LIN {X 0,Y 404.174,Z 269.949,A -85,B 0,C 180,E1 -11024.526,E2 -11024.526} C_VEL
LIN {X 0,Y 404.186,Z 269.95,A -85,B 0,C 180,E1 -11027.302,E2 -11027.302} C_VEL
LIN {X 0,Y 404.143,Z 269.956,A -85,B 0,C 180,E1 -11029.952,E2 -11029.952} C_VEL
LIN {X 0,Y 404.113,Z 269.963,A -85,B 0,C 180,E1 -11033.121,E2 -11033.121} C_VEL
LIN {X 0,Y 404.144,Z 270.047,A -85,B 0,C 180,E1 -11034.335,E2 -11034.335} C_VEL
LIN {X 0,Y 405.121,Z 276.124,A -85,B 0,C 180,E1 -11035.981,E2 -11035.981} C_VEL
LIN {X 0,Y 405.001,Z 280.687,A -85,B 0,C 180,E1 -11037.137,E2 -11037.137} C_VEL
LIN {X 0,Y 408.445,Z 296.726,A -85,B 0,C 180,E1 -11037.6,E2 -11037.6} C_VEL
LIN {X 0,Y 407.757,Z 357.433,A -85,B 0,C 180,E1 -11038.715,E2 -11038.715} C_VEL
LIN {X 0,Y 407.545,Z 367.165,A -85,B 0,C 180,E1 -11039.032,E2 -11039.032} C_VEL
LIN {X 0,Y 407.188,Z 378.033,A -85,B 0,C 180,E1 -11039.56,E2 -11039.56} C_VEL
LIN {X 0,Y 406.752,Z 387.643,A -85,B 0,C 180,E1 -11040.215,E2 -11040.215} C_VEL
LIN {X 0,Y 406.183,Z 396.777,A -85,B 0,C 180,E1 -11041.022,E2 -11041.022} C_VEL
LIN {X 0,Y 405.632,Z 404.168,A -85,B 0,C 180,E1 -11041.827,E2 -11041.827} C_VEL
LIN {X 0,Y 405.183,Z 410.356,A -85,B 0,C 180,E1 -11042.636,E2 -11042.636} C_VEL
LIN {X 0,Y 404.65,Z 417.143,A -85,B 0,C 180,E1 -11043.712,E2 -11043.712} C_VEL
LIN {X 0,Y 404.296,Z 422.137,A -85,B 0,C 180,E1 -11044.668,E2 -11044.668} C_VEL
LIN {X 0,Y 403.869,Z 427.256,A -85,B 0,C 180,E1 -11045.862,E2 -11045.862} C_VEL
LIN {X 0,Y 403.556,Z 430.963,A -85,B 0,C 180,E1 -11046.932,E2 -11046.932} C_VEL
LIN {X 0,Y 403.244,Z 435.139,A -85,B 0,C 180,E1 -11048.531,E2 -11048.531} C_VEL
LIN {X 0,Y 402.977,Z 438.166,A -85,B 0,C 180,E1 -11050.336,E2 -11050.336} C_VEL
LIN {X 0,Y 402.842,Z 439.29,A -85,B 0,C 180,E1 -11051.698,E2 -11051.698} C_VEL
LIN {X 0,Y 402.817,Z 439.578,A -85,B 0,C 180,E1 -11052.747,E2 -11052.747} C_VEL
LIN {X 0,Y 402.872,Z 439.249,A -85,B 0,C 180,E1 -11053.793,E2 -11053.793} C_VEL
LIN {X 0,Y 402.868,Z 438.387,A -85,B 0,C 180,E1 -11054.831,E2 -11054.831} C_VEL
LIN {X 0,Y 402.939,Z 437.007,A -85,B 0,C 180,E1 -11055.866,E2 -11055.866} C_VEL
LIN {X 0,Y 403.162,Z 433.812,A -85,B 0,C 180,E1 -11057.451,E2 -11057.451} C_VEL
LIN {X 0,Y 403.373,Z 429.458,A -85,B 0,C 180,E1 -11058.951,E2 -11058.951} C_VEL
LIN {X 0,Y 403.667,Z 424.469,A -85,B 0,C 180,E1 -11060.227,E2 -11060.227} C_VEL
LIN {X 0,Y 404.026,Z 418.153,A -85,B 0,C 180,E1 -11061.497,E2 -11061.497} C_VEL
LIN {X 0,Y 404.338,Z 412.472,A -85,B 0,C 180,E1 -11062.437,E2 -11062.437} C_VEL
LIN {X 0,Y 404.715,Z 405.485,A -85,B 0,C 180,E1 -11063.394,E2 -11063.394} C_VEL
LIN {X 0,Y 405.091,Z 398.855,A -85,B 0,C 180,E1 -11064.15,E2 -11064.15} C_VEL
LIN {X 0,Y 405.519,Z 390.81,A -85,B 0,C 180,E1 -11064.904,E2 -11064.904} C_VEL
LIN {X 0,Y 405.865,Z 382.508,A -85,B 0,C 180,E1 -11065.531,E2 -11065.531} C_VEL
LIN {X 0,Y 406.085,Z 374.124,A -85,B 0,C 180,E1 -11066.031,E2 -11066.031} C_VEL
LIN {X 0,Y 406.347,Z 364.962,A -85,B 0,C 180,E1 -11066.437,E2 -11066.437} C_VEL
LIN {X 0,Y 406.545,Z 355.549,A -85,B 0,C 180,E1 -11066.717,E2 -11066.717} C_VEL
LIN {X 0,Y 406.925,Z 321.203,A -85,B 0,C 180,E1 -11067.342,E2 -11067.342} C_VEL
LIN {X 0,Y 406.415,Z 315.379,A -85,B 0,C 180,E1 -11067.462,E2 -11067.462} C_VEL
LIN {X 0,Y 403.768,Z 306.003,A -85,B 0,C 180,E1 -11067.712,E2 -11067.712} C_VEL
LIN {X 0,Y 401.116,Z 298.58,A -85,B 0,C 180,E1 -11067.929,E2 -11067.929} C_VEL
LIN {X 0,Y 399.043,Z 290.982,A -85,B 0,C 180,E1 -11068.133,E2 -11068.133} C_VEL
LIN {X 0,Y 397.37,Z 280.75,A -85,B 0,C 180,E1 -11068.385,E2 -11068.385} C_VEL
LIN {X 0,Y 397.583,Z 272.725,A -85,B 0,C 180,E1 -11070.507,E2 -11070.507} C_VEL
LIN {X 0,Y 397.366,Z 270.803,A -85,B 0,C 180,E1 -11071.077,E2 -11071.077} C_VEL
LIN {X 0,Y 397.345,Z 270.804,A -85,B 0,C 180,E1 -11073.042,E2 -11073.042} C_VEL
LIN {X 0,Y 397.319,Z 270.807,A -85,B 0,C 180,E1 -11077.113,E2 -11077.113} C_VEL
LIN {X 0,Y 397.182,Z 270.819,A -85,B 0,C 180,E1 -11080.192,E2 -11080.192} C_VEL
LIN {X 0,Y 397.192,Z 270.825,A -85,B 0,C 180,E1 -11083.322,E2 -11083.322} C_VEL
LIN {X 0,Y 397.148,Z 270.828,A -85,B 0,C 180,E1 -11087.157,E2 -11087.157} C_VEL
LIN {X 0,Y 397.075,Z 270.833,A -85,B 0,C 180,E1 -11090.732,E2 -11090.732} C_VEL
LIN {X 0,Y 397.091,Z 270.831,A -85,B 0,C 180,E1 -11094.021,E2 -11094.021} C_VEL
LIN {X 0,Y 397.061,Z 270.837,A -85,B 0,C 180,E1 -11097.759,E2 -11097.759} C_VEL
LIN {X 0,Y 397.048,Z 270.836,A -85,B 0,C 180,E1 -11100.885,E2 -11100.885} C_VEL
LIN {X 0,Y 397.097,Z 270.829,A -85,B 0,C 180,E1 -11104.496,E2 -11104.496} C_VEL
LIN {X 0,Y 397.065,Z 270.834,A -85,B 0,C 180,E1 -11108.28,E2 -11108.28} C_VEL
LIN {X 0,Y 397.033,Z 270.841,A -85,B 0,C 180,E1 -11111.981,E2 -11111.981} C_VEL
LIN {X 0,Y 397.064,Z 270.835,A -85,B 0,C 180,E1 -11115.073,E2 -11115.073} C_VEL
LIN {X 0,Y 397.045,Z 270.839,A -85,B 0,C 180,E1 -11118.025,E2 -11118.025} C_VEL
LIN {X 0,Y 397.106,Z 270.829,A -85,B 0,C 180,E1 -11121.143,E2 -11121.143} C_VEL
LIN {X 0,Y 397.102,Z 270.83,A -85,B 0,C 180,E1 -11124.501,E2 -11124.501} C_VEL
LIN {X 0,Y 397.064,Z 270.84,A -85,B 0,C 180,E1 -11127.932,E2 -11127.932} C_VEL
LIN {X 0,Y 397.105,Z 270.831,A -85,B 0,C 180,E1 -11130.299,E2 -11130.299} C_VEL
LIN {X 0,Y 397.083,Z 270.836,A -85,B 0,C 180,E1 -11133.743,E2 -11133.743} C_VEL
LIN {X 0,Y 397.094,Z 270.831,A -85,B 0,C 180,E1 -11137.089,E2 -11137.089} C_VEL
LIN {X 0,Y 397.141,Z 270.827,A -85,B 0,C 180,E1 -11140.357,E2 -11140.357} C_VEL
LIN {X 0,Y 397.248,Z 270.921,A -85,B 0,C 180,E1 -11142.721,E2 -11142.721} C_VEL
LIN {X 0,Y 397.144,Z 279.933,A -85,B 0,C 180,E1 -11145.005,E2 -11145.005} C_VEL
LIN {X 0,Y 399.627,Z 297.894,A -85,B 0,C 180,E1 -11145.49,E2 -11145.49} C_VEL
LIN {X 0,Y 398.723,Z 357.712,A -85,B 0,C 180,E1 -11146.855,E2 -11146.855} C_VEL
LIN {X 0,Y 398.525,Z 367.209,A -85,B 0,C 180,E1 -11147.204,E2 -11147.204} C_VEL
LIN {X 0,Y 398.257,Z 377.066,A -85,B 0,C 180,E1 -11147.713,E2 -11147.713} C_VEL
LIN {X 0,Y 397.95,Z 387.333,A -85,B 0,C 180,E1 -11148.415,E2 -11148.415} C_VEL
LIN {X 0,Y 397.542,Z 397.262,A -85,B 0,C 180,E1 -11149.306,E2 -11149.306} C_VEL
LIN {X 0,Y 397.235,Z 405.182,A -85,B 0,C 180,E1 -11150.199,E2 -11150.199} C_VEL
LIN {X 0,Y 396.884,Z 411.771,A -85,B 0,C 180,E1 -11151.09,E2 -11151.09} C_VEL
LIN {X 0,Y 396.59,Z 418.055,A -85,B 0,C 180,E1 -11152.11,E2 -11152.11} C_VEL
LIN {X 0,Y 396.441,Z 423.135,A -85,B 0,C 180,E1 -11153.1,E2 -11153.1} C_VEL
LIN {X 0,Y 396.217,Z 428.598,A -85,B 0,C 180,E1 -11154.405,E2 -11154.405} C_VEL
LIN {X 0,Y 396.034,Z 433.483,A -85,B 0,C 180,E1 -11155.933,E2 -11155.933} C_VEL
LIN {X 0,Y 395.981,Z 435.892,A -85,B 0,C 180,E1 -11156.951,E2 -11156.951} C_VEL
LIN {X 0,Y 395.905,Z 437.67,A -85,B 0,C 180,E1 -11157.969,E2 -11157.969} C_VEL
LIN {X 0,Y 395.839,Z 438.894,A -85,B 0,C 180,E1 -11158.986,E2 -11158.986} C_VEL
LIN {X 0,Y 395.826,Z 439.592,A -85,B 0,C 180,E1 -11160.003,E2 -11160.003} C_VEL
LIN {X 0,Y 395.863,Z 439.772,A -85,B 0,C 180,E1 -11161.02,E2 -11161.02} C_VEL
LIN {X 0,Y 395.955,Z 439.429,A -85,B 0,C 180,E1 -11162.038,E2 -11162.038} C_VEL
LIN {X 0,Y 396.117,Z 438.507,A -85,B 0,C 180,E1 -11163.054,E2 -11163.054} C_VEL
LIN {X 0,Y 396.429,Z 436.049,A -85,B 0,C 180,E1 -11164.579,E2 -11164.579} C_VEL
LIN {X 0,Y 396.518,Z 433.747,A -85,B 0,C 180,E1 -11165.597,E2 -11165.597} C_VEL
LIN {X 0,Y 396.712,Z 430.771,A -85,B 0,C 180,E1 -11166.615,E2 -11166.615} C_VEL
LIN {X 0,Y 397.14,Z 426.848,A -85,B 0,C 180,E1 -11167.688,E2 -11167.688} C_VEL
LIN {X 0,Y 397.653,Z 420.011,A -85,B 0,C 180,E1 -11169.155,E2 -11169.155} C_VEL
LIN {X 0,Y 398.088,Z 414.112,A -85,B 0,C 180,E1 -11170.171,E2 -11170.171} C_VEL
LIN {X 0,Y 398.67,Z 406.947,A -85,B 0,C 180,E1 -11171.184,E2 -11171.184} C_VEL
LIN {X 0,Y 399.293,Z 398.187,A -85,B 0,C 180,E1 -11172.196,E2 -11172.196} C_VEL
LIN {X 0,Y 399.921,Z 388.436,A -85,B 0,C 180,E1 -11173.08,E2 -11173.08} C_VEL
LIN {X 0,Y 400.428,Z 378.521,A -85,B 0,C 180,E1 -11173.774,E2 -11173.774} C_VEL
LIN {X 0,Y 400.814,Z 369.089,A -85,B 0,C 180,E1 -11174.278,E2 -11174.278} C_VEL
LIN {X 0,Y 401.151,Z 358.396,A -85,B 0,C 180,E1 -11174.687,E2 -11174.687} C_VEL
LIN {X 0,Y 402.704,Z 298.527,A -85,B 0,C 180,E1 -11176.176,E2 -11176.176} C_VEL
LIN {X 0,Y 399.798,Z 286.257,A -85,B 0,C 180,E1 -11176.72,E2 -11176.72} C_VEL
LIN {X 0,Y 398.727,Z 282.083,A -85,B 0,C 180,E1 -11176.943,E2 -11176.943} C_VEL
LIN {X 0,Y 398.602,Z 277.725,A -85,B 0,C 180,E1 -11178.064,E2 -11178.064} C_VEL
LIN {X 0,Y 397.171,Z 270.829,A -85,B 0,C 180,E1 -11179.972,E2 -11179.972} C_VEL
LIN {X 0,Y 397.127,Z 270.833,A -85,B 0,C 180,E1 -11184.021,E2 -11184.021} C_VEL
LIN {X 0,Y 397.102,Z 270.834,A -85,B 0,C 180,E1 -11187.759,E2 -11187.759} C_VEL
LIN {X 0,Y 397.087,Z 270.836,A -85,B 0,C 180,E1 -11190.884,E2 -11190.884} C_VEL
LIN {X 0,Y 397.126,Z 270.832,A -85,B 0,C 180,E1 -11194.496,E2 -11194.496} C_VEL
LIN {X 0,Y 397.101,Z 270.834,A -85,B 0,C 180,E1 -11198.278,E2 -11198.278} C_VEL
LIN {X 0,Y 397.067,Z 270.837,A -85,B 0,C 180,E1 -11201.979,E2 -11201.979} C_VEL
LIN {X 0,Y 397.096,Z 270.832,A -85,B 0,C 180,E1 -11205.07,E2 -11205.07} C_VEL
LIN {X 0,Y 397.07,Z 270.834,A -85,B 0,C 180,E1 -11208.023,E2 -11208.023} C_VEL
LIN {X 0,Y 397.109,Z 270.831,A -85,B 0,C 180,E1 -11211.145,E2 -11211.145} C_VEL
LIN {X 0,Y 397.125,Z 270.83,A -85,B 0,C 180,E1 -11214.498,E2 -11214.498} C_VEL
LIN {X 0,Y 397.086,Z 270.834,A -85,B 0,C 180,E1 -11217.929,E2 -11217.929} C_VEL
LIN {X 0,Y 397.131,Z 270.829,A -85,B 0,C 180,E1 -11221.457,E2 -11221.457} C_VEL
LIN {X 0,Y 397.233,Z 270.885,A -85,B 0,C 180,E1 -11224.416,E2 -11224.416} C_VEL
LIN {X 0,Y 398.807,Z 280.938,A -85,B 0,C 180,E1 -11226.824,E2 -11226.824} C_VEL
LIN {X 0,Y 398.07,Z 294.332,A -85,B 0,C 180,E1 -11229.862,E2 -11229.862} C_VEL
LIN {X 0,Y 397.236,Z 309.12,A -85,B 0,C 180,E1 -11233.183,E2 -11233.183} C_VEL
LIN {X 0,Y 400.225,Z 328.076,A -85,B 0,C 180,E1 -11233.934,E2 -11233.934} C_VEL
LIN {X 0,Y 401.508,Z 342.829,A -85,B 0,C 180,E1 -11234.415,E2 -11234.415} C_VEL
LIN {X 0,Y 400.145,Z 395.197,A -85,B 0,C 180,E1 -11235.739,E2 -11235.739} C_VEL
LIN {X 0,Y 399.501,Z 407.511,A -85,B 0,C 180,E1 -11236.261,E2 -11236.261} C_VEL
LIN {X 0,Y 399.004,Z 415.953,A -85,B 0,C 180,E1 -11236.763,E2 -11236.763} C_VEL
LIN {X 0,Y 398.483,Z 424.385,A -85,B 0,C 180,E1 -11237.393,E2 -11237.393} C_VEL
LIN {X 0,Y 397.952,Z 432.588,A -85,B 0,C 180,E1 -11238.153,E2 -11238.153} C_VEL
LIN {X 0,Y 397.399,Z 440.44,A -85,B 0,C 180,E1 -11239.04,E2 -11239.04} C_VEL
LIN {X 0,Y 396.78,Z 449.471,A -85,B 0,C 180,E1 -11240.313,E2 -11240.313} C_VEL
LIN {X 0,Y 396.386,Z 456.463,A -85,B 0,C 180,E1 -11241.589,E2 -11241.589} C_VEL
LIN {X 0,Y 396.123,Z 462.075,A -85,B 0,C 180,E1 -11242.866,E2 -11242.866} C_VEL
LIN {X 0,Y 395.87,Z 467.423,A -85,B 0,C 180,E1 -11244.396,E2 -11244.396} C_VEL
LIN {X 0,Y 395.822,Z 471.467,A -85,B 0,C 180,E1 -11245.927,E2 -11245.927} C_VEL
LIN {X 0,Y 395.822,Z 473.455,A -85,B 0,C 180,E1 -11246.946,E2 -11246.946} C_VEL
LIN {X 0,Y 395.887,Z 474.938,A -85,B 0,C 180,E1 -11247.965,E2 -11247.965} C_VEL
LIN {X 0,Y 395.835,Z 475.884,A -85,B 0,C 180,E1 -11248.982,E2 -11248.982} C_VEL
LIN {X 0,Y 395.824,Z 476.239,A -85,B 0,C 180,E1 -11250,E2 -11250} C_VEL
LIN {X 0,Y 395.825,Z 476.118,A -85,B 0,C 180,E1 -11251.017,E2 -11251.017} C_VEL
LIN {X 0,Y 395.863,Z 475.535,A -85,B 0,C 180,E1 -11252.035,E2 -11252.035} C_VEL
LIN {X 0,Y 395.785,Z 474.474,A -85,B 0,C 180,E1 -11253.053,E2 -11253.053} C_VEL
LIN {X 0,Y 395.881,Z 471.773,A -85,B 0,C 180,E1 -11254.582,E2 -11254.582} C_VEL
LIN {X 0,Y 395.873,Z 469.352,A -85,B 0,C 180,E1 -11255.603,E2 -11255.603} C_VEL
LIN {X 0,Y 396.138,Z 464.417,A -85,B 0,C 180,E1 -11257.134,E2 -11257.134} C_VEL
LIN {X 0,Y 396.439,Z 459.13,A -85,B 0,C 180,E1 -11258.41,E2 -11258.41} C_VEL
LIN {X 0,Y 396.839,Z 453.959,A -85,B 0,C 180,E1 -11259.428,E2 -11259.428} C_VEL
LIN {X 0,Y 397.316,Z 447.75,A -85,B 0,C 180,E1 -11260.446,E2 -11260.446} C_VEL
LIN {X 0,Y 397.808,Z 441.234,A -85,B 0,C 180,E1 -11261.335,E2 -11261.335} C_VEL
LIN {X 0,Y 398.374,Z 433.361,A -85,B 0,C 180,E1 -11262.222,E2 -11262.222} C_VEL
LIN {X 0,Y 399.005,Z 425.058,A -85,B 0,C 180,E1 -11262.978,E2 -11262.978} C_VEL
LIN {X 0,Y 399.684,Z 414.494,A -85,B 0,C 180,E1 -11263.732,E2 -11263.732} C_VEL
LIN {X 0,Y 400.244,Z 402.924,A -85,B 0,C 180,E1 -11264.303,E2 -11264.303} C_VEL
LIN {X 0,Y 400.662,Z 393.87,A -85,B 0,C 180,E1 -11264.601,E2 -11264.601} C_VEL
LIN {X 0,Y 401.065,Z 364.271,A -85,B 0,C 180,E1 -11265.172,E2 -11265.172} C_VEL
LIN {X 0,Y 401.215,Z 341.462,A -85,B 0,C 180,E1 -11265.592,E2 -11265.592} C_VEL
LIN {X 0,Y 399.203,Z 325.467,A -85,B 0,C 180,E1 -11265.99,E2 -11265.99} C_VEL
LIN {X 0,Y 397.495,Z 314.886,A -85,B 0,C 180,E1 -11266.295,E2 -11266.295} C_VEL
LIN {X 0,Y 398.489,Z 298.029,A -85,B 0,C 180,E1 -11270.115,E2 -11270.115} C_VEL
LIN {X 0,Y 399.419,Z 284.203,A -85,B 0,C 180,E1 -11273.296,E2 -11273.296} C_VEL
LIN {X 0,Y 398.417,Z 277.116,A -85,B 0,C 180,E1 -11275.046,E2 -11275.046} C_VEL
LIN {X 0,Y 397.187,Z 270.824,A -85,B 0,C 180,E1 -11276.679,E2 -11276.679} C_VEL
LIN {X 0,Y 397.109,Z 270.829,A -85,B 0,C 180,E1 -11279.863,E2 -11279.863} C_VEL
LIN {X 0,Y 397.119,Z 270.83,A -85,B 0,C 180,E1 -11283.272,E2 -11283.272} C_VEL
LIN {X 0,Y 397.104,Z 270.829,A -85,B 0,C 180,E1 -11286.994,E2 -11286.994} C_VEL
LIN {X 0,Y 397.085,Z 270.833,A -85,B 0,C 180,E1 -11290.44,E2 -11290.44} C_VEL
LIN {X 0,Y 397.108,Z 270.831,A -85,B 0,C 180,E1 -11293.647,E2 -11293.647} C_VEL
LIN {X 0,Y 397.108,Z 270.829,A -85,B 0,C 180,E1 -11296.52,E2 -11296.52} C_VEL
LIN {X 0,Y 397.094,Z 270.828,A -85,B 0,C 180,E1 -11300.418,E2 -11300.418} C_VEL
LIN {X 0,Y 397.104,Z 270.83,A -85,B 0,C 180,E1 -11303.003,E2 -11303.003} C_VEL
LIN {X 0,Y 397.125,Z 270.827,A -85,B 0,C 180,E1 -11306.28,E2 -11306.28} C_VEL
LIN {X 0,Y 397.107,Z 270.831,A -85,B 0,C 180,E1 -11310.135,E2 -11310.135} C_VEL
LIN {X 0,Y 397.102,Z 270.829,A -85,B 0,C 180,E1 -11313.737,E2 -11313.737} C_VEL
LIN {X 0,Y 397.11,Z 270.829,A -85,B 0,C 180,E1 -11317.083,E2 -11317.083} C_VEL
LIN {X 0,Y 397.152,Z 270.824,A -85,B 0,C 180,E1 -11320.35,E2 -11320.35} C_VEL
LIN {X 0,Y 397.171,Z 270.818,A -85,B 0,C 180,E1 -11323.551,E2 -11323.551} C_VEL
LIN {X 0,Y 397.233,Z 270.811,A -85,B 0,C 180,E1 -11326.7,E2 -11326.7} C_VEL
LIN {X 0,Y 397.22,Z 270.809,A -85,B 0,C 180,E1 -11329.806,E2 -11329.806} C_VEL
LIN {X 0,Y 397.352,Z 270.793,A -85,B 0,C 180,E1 -11332.885,E2 -11332.885} C_VEL
LIN {X 0,Y 397.25,Z 270.802,A -85,B 0,C 180,E1 -11334.922,E2 -11334.922} C_VEL
LIN {X 0,Y 397.446,Z 270.789,A -85,B 0,C 180,E1 -11337.97,E2 -11337.97} C_VEL
LIN {X 0,Y 397.575,Z 270.765,A -85,B 0,C 180,E1 -11339.997,E2 -11339.997} C_VEL
LIN {X 0,Y 397.367,Z 270.794,A -85,B 0,C 180,E1 -11343.038,E2 -11343.038} C_VEL
LIN {X 0,Y 397.314,Z 270.798,A -85,B 0,C 180,E1 -11346.518,E2 -11346.518} C_VEL
LIN {X 0,Y 397.232,Z 270.811,A -85,B 0,C 180,E1 -11349.159,E2 -11349.159} C_VEL
LIN {X 0,Y 397.214,Z 270.818,A -85,B 0,C 180,E1 -11352.254,E2 -11352.254} C_VEL
LIN {X 0,Y 397.172,Z 270.816,A -85,B 0,C 180,E1 -11355.388,E2 -11355.388} C_VEL
LIN {X 0,Y 397.152,Z 270.826,A -85,B 0,C 180,E1 -11358.57,E2 -11358.57} C_VEL
LIN {X 0,Y 397.086,Z 270.831,A -85,B 0,C 180,E1 -11361.815,E2 -11361.815} C_VEL
LIN {X 0,Y 397.144,Z 270.823,A -85,B 0,C 180,E1 -11365.128,E2 -11365.128} C_VEL
LIN {X 0,Y 397.148,Z 270.824,A -85,B 0,C 180,E1 -11367.772,E2 -11367.772} C_VEL
LIN {X 0,Y 397.063,Z 270.835,A -85,B 0,C 180,E1 -11370.879,E2 -11370.879} C_VEL
LIN {X 0,Y 397.108,Z 270.829,A -85,B 0,C 180,E1 -11374.49,E2 -11374.49} C_VEL
LIN {X 0,Y 397.082,Z 270.836,A -85,B 0,C 180,E1 -11378.272,E2 -11378.272} C_VEL
LIN {X 0,Y 397.132,Z 270.828,A -85,B 0,C 180,E1 -11381.989,E2 -11381.989} C_VEL
LIN {X 0,Y 397.127,Z 270.832,A -85,B 0,C 180,E1 -11385.056,E2 -11385.056} C_VEL
LIN {X 0,Y 397.131,Z 270.828,A -85,B 0,C 180,E1 -11388.004,E2 -11388.004} C_VEL
LIN {X 0,Y 397.083,Z 270.837,A -85,B 0,C 180,E1 -11391.723,E2 -11391.723} C_VEL
LIN {X 0,Y 397.145,Z 271.028,A -85,B 0,C 180,E1 -11394.113,E2 -11394.113} C_VEL
LIN {X 0,Y 398.139,Z 276.42,A -85,B 0,C 180,E1 -11395.607,E2 -11395.607} C_VEL
LIN {X 0,Y 398.069,Z 280.908,A -85,B 0,C 180,E1 -11396.78,E2 -11396.78} C_VEL
LIN {X 0,Y 401.763,Z 297.882,A -85,B 0,C 180,E1 -11397.299,E2 -11397.299} C_VEL
LIN {X 0,Y 401.021,Z 356.746,A -85,B 0,C 180,E1 -11398.392,E2 -11398.392} C_VEL
LIN {X 0,Y 400.847,Z 365.689,A -85,B 0,C 180,E1 -11398.671,E2 -11398.671} C_VEL
LIN {X 0,Y 400.555,Z 374.511,A -85,B 0,C 180,E1 -11399.071,E2 -11399.071} C_VEL
LIN {X 0,Y 400.146,Z 383.219,A -85,B 0,C 180,E1 -11399.599,E2 -11399.599} C_VEL
LIN {X 0,Y 399.581,Z 392.811,A -85,B 0,C 180,E1 -11400.352,E2 -11400.352} C_VEL
LIN {X 0,Y 398.882,Z 403.425,A -85,B 0,C 180,E1 -11401.45,E2 -11401.45} C_VEL
LIN {X 0,Y 398.239,Z 410.921,A -85,B 0,C 180,E1 -11402.44,E2 -11402.44} C_VEL
LIN {X 0,Y 397.704,Z 417.477,A -85,B 0,C 180,E1 -11403.5,E2 -11403.5} C_VEL
LIN {X 0,Y 397.298,Z 422.771,A -85,B 0,C 180,E1 -11404.538,E2 -11404.538} C_VEL
LIN {X 0,Y 396.886,Z 427.59,A -85,B 0,C 180,E1 -11405.688,E2 -11405.688} C_VEL
LIN {X 0,Y 396.461,Z 432.093,A -85,B 0,C 180,E1 -11407.046,E2 -11407.046} C_VEL
LIN {X 0,Y 396.245,Z 434.867,A -85,B 0,C 180,E1 -11408.132,E2 -11408.132} C_VEL
LIN {X 0,Y 396.046,Z 436.997,A -85,B 0,C 180,E1 -11409.212,E2 -11409.212} C_VEL
LIN {X 0,Y 395.903,Z 438.541,A -85,B 0,C 180,E1 -11410.289,E2 -11410.289} C_VEL
LIN {X 0,Y 395.786,Z 439.51,A -85,B 0,C 180,E1 -11411.36,E2 -11411.36} C_VEL
LIN {X 0,Y 395.742,Z 439.857,A -85,B 0,C 180,E1 -11412.428,E2 -11412.428} C_VEL
LIN {X 0,Y 395.753,Z 439.659,A -85,B 0,C 180,E1 -11413.51,E2 -11413.51} C_VEL
LIN {X 0,Y 395.784,Z 438.964,A -85,B 0,C 180,E1 -11414.553,E2 -11414.553} C_VEL
LIN {X 0,Y 395.846,Z 437.749,A -85,B 0,C 180,E1 -11415.608,E2 -11415.608} C_VEL
LIN {X 0,Y 395.968,Z 435.998,A -85,B 0,C 180,E1 -11416.66,E2 -11416.66} C_VEL
LIN {X 0,Y 396.168,Z 432.139,A -85,B 0,C 180,E1 -11418.229,E2 -11418.229} C_VEL
LIN {X 0,Y 396.47,Z 426.872,A -85,B 0,C 180,E1 -11419.79,E2 -11419.79} C_VEL
LIN {X 0,Y 396.799,Z 421.208,A -85,B 0,C 180,E1 -11421.085,E2 -11421.085} C_VEL
LIN {X 0,Y 397.254,Z 413.626,A -85,B 0,C 180,E1 -11422.432,E2 -11422.432} C_VEL
LIN {X 0,Y 397.692,Z 405.791,A -85,B 0,C 180,E1 -11423.532,E2 -11423.532} C_VEL
LIN {X 0,Y 398.08,Z 399.158,A -85,B 0,C 180,E1 -11424.301,E2 -11424.301} C_VEL
LIN {X 0,Y 398.533,Z 391.104,A -85,B 0,C 180,E1 -11425.068,E2 -11425.068} C_VEL
LIN {X 0,Y 398.879,Z 382.802,A -85,B 0,C 180,E1 -11425.706,E2 -11425.706} C_VEL
LIN {X 0,Y 399.122,Z 374.4,A -85,B 0,C 180,E1 -11426.214,E2 -11426.214} C_VEL
LIN {X 0,Y 399.395,Z 365.22,A -85,B 0,C 180,E1 -11426.627,E2 -11426.627} C_VEL
LIN {X 0,Y 399.598,Z 355.776,A -85,B 0,C 180,E1 -11426.913,E2 -11426.913} C_VEL
LIN {X 0,Y 400.109,Z 296.595,A -85,B 0,C 180,E1 -11427.997,E2 -11427.997} C_VEL
LIN {X 0,Y 399.043,Z 290.982,A -85,B 0,C 180,E1 -11428.133,E2 -11428.133} C_VEL
LIN {X 0,Y 397.721,Z 287.251,A -85,B 0,C 180,E1 -11428.29,E2 -11428.29} C_VEL
LIN {X 0,Y 394.97,Z 283.108,A -85,B 0,C 180,E1 -11428.648,E2 -11428.648} C_VEL
LIN {X 0,Y 392.229,Z 279.677,A -85,B 0,C 180,E1 -11429.148,E2 -11429.148} C_VEL
LIN {X 0,Y 390.853,Z 277.401,A -85,B 0,C 180,E1 -11429.612,E2 -11429.612} C_VEL
LIN {X 0,Y 390.591,Z 276.013,A -85,B 0,C 180,E1 -11429.956,E2 -11429.956} C_VEL
LIN {X 0,Y 390.337,Z 271.679,A -85,B 0,C 180,E1 -11431.161,E2 -11431.161} C_VEL
LIN {X 0,Y 390.279,Z 271.685,A -85,B 0,C 180,E1 -11433.097,E2 -11433.097} C_VEL
LIN {X 0,Y 390.29,Z 271.678,A -85,B 0,C 180,E1 -11436.203,E2 -11436.203} C_VEL
LIN {X 0,Y 390.169,Z 271.699,A -85,B 0,C 180,E1 -11439.33,E2 -11439.33} C_VEL
LIN {X 0,Y 390.16,Z 271.699,A -85,B 0,C 180,E1 -11443.44,E2 -11443.44} C_VEL
LIN {X 0,Y 390.115,Z 271.706,A -85,B 0,C 180,E1 -11447.309,E2 -11447.309} C_VEL
LIN {X 0,Y 390.055,Z 271.707,A -85,B 0,C 180,E1 -11450.472,E2 -11450.472} C_VEL
LIN {X 0,Y 390.034,Z 271.715,A -85,B 0,C 180,E1 -11453.355,E2 -11453.355} C_VEL
LIN {X 0,Y 390.023,Z 271.711,A -85,B 0,C 180,E1 -11456.775,E2 -11456.775} C_VEL
LIN {X 0,Y 390.007,Z 271.713,A -85,B 0,C 180,E1 -11460.303,E2 -11460.303} C_VEL
LIN {X 0,Y 390.041,Z 271.71,A -85,B 0,C 180,E1 -11464.028,E2 -11464.028} C_VEL
LIN {X 0,Y 390.013,Z 271.719,A -85,B 0,C 180,E1 -11467.553,E2 -11467.553} C_VEL
LIN {X 0,Y 389.994,Z 271.714,A -85,B 0,C 180,E1 -11470.818,E2 -11470.818} C_VEL
LIN {X 0,Y 390.031,Z 271.714,A -85,B 0,C 180,E1 -11473.889,E2 -11473.889} C_VEL
LIN {X 0,Y 390.036,Z 271.709,A -85,B 0,C 180,E1 -11476.793,E2 -11476.793} C_VEL
LIN {X 0,Y 390.037,Z 271.714,A -85,B 0,C 180,E1 -11479.564,E2 -11479.564} C_VEL
LIN {X 0,Y 390.024,Z 271.712,A -85,B 0,C 180,E1 -11482.454,E2 -11482.454} C_VEL
LIN {X 0,Y 390.052,Z 271.711,A -85,B 0,C 180,E1 -11486.049,E2 -11486.049} C_VEL
LIN {X 0,Y 390.031,Z 271.717,A -85,B 0,C 180,E1 -11489.874,E2 -11489.874} C_VEL
LIN {X 0,Y 390.043,Z 271.709,A -85,B 0,C 180,E1 -11493.231,E2 -11493.231} C_VEL
LIN {X 0,Y 390.058,Z 271.707,A -85,B 0,C 180,E1 -11496.768,E2 -11496.768} C_VEL
LIN {X 0,Y 390.097,Z 271.708,A -85,B 0,C 180,E1 -11499.987,E2 -11499.987} C_VEL
LIN {X 0,Y 390.195,Z 271.716,A -85,B 0,C 180,E1 -11502.672,E2 -11502.672} C_VEL
LIN {X 0,Y 390.118,Z 280.193,A -85,B 0,C 180,E1 -11504.833,E2 -11504.833} C_VEL
LIN {X 0,Y 392.636,Z 298.37,A -85,B 0,C 180,E1 -11505.333,E2 -11505.333} C_VEL
LIN {X 0,Y 391.685,Z 358.471,A -85,B 0,C 180,E1 -11506.746,E2 -11506.746} C_VEL
LIN {X 0,Y 391.423,Z 369.194,A -85,B 0,C 180,E1 -11507.166,E2 -11507.166} C_VEL
LIN {X 0,Y 391.103,Z 379.735,A -85,B 0,C 180,E1 -11507.749,E2 -11507.749} C_VEL
LIN {X 0,Y 390.777,Z 390.845,A -85,B 0,C 180,E1 -11508.594,E2 -11508.594} C_VEL
LIN {X 0,Y 390.45,Z 398.893,A -85,B 0,C 180,E1 -11509.372,E2 -11509.372} C_VEL
LIN {X 0,Y 390.113,Z 406.617,A -85,B 0,C 180,E1 -11510.28,E2 -11510.28} C_VEL
LIN {X 0,Y 389.683,Z 414.751,A -85,B 0,C 180,E1 -11511.447,E2 -11511.447} C_VEL
LIN {X 0,Y 389.457,Z 421.9,A -85,B 0,C 180,E1 -11512.747,E2 -11512.747} C_VEL
LIN {X 0,Y 389.186,Z 426.546,A -85,B 0,C 180,E1 -11513.783,E2 -11513.783} C_VEL
LIN {X 0,Y 389.099,Z 430.404,A -85,B 0,C 180,E1 -11514.822,E2 -11514.822} C_VEL
LIN {X 0,Y 388.953,Z 433.537,A -85,B 0,C 180,E1 -11515.859,E2 -11515.859} C_VEL
LIN {X 0,Y 388.887,Z 435.986,A -85,B 0,C 180,E1 -11516.896,E2 -11516.896} C_VEL
LIN {X 0,Y 388.823,Z 437.826,A -85,B 0,C 180,E1 -11517.932,E2 -11517.932} C_VEL
LIN {X 0,Y 388.769,Z 439.122,A -85,B 0,C 180,E1 -11518.968,E2 -11518.968} C_VEL
LIN {X 0,Y 388.753,Z 439.893,A -85,B 0,C 180,E1 -11520.003,E2 -11520.003} C_VEL
LIN {X 0,Y 388.792,Z 440.148,A -85,B 0,C 180,E1 -11521.039,E2 -11521.039} C_VEL
LIN {X 0,Y 388.891,Z 439.859,A -85,B 0,C 180,E1 -11522.075,E2 -11522.075} C_VEL
LIN {X 0,Y 389.064,Z 438.964,A -85,B 0,C 180,E1 -11523.11,E2 -11523.11} C_VEL
LIN {X 0,Y 389.393,Z 436.637,A -85,B 0,C 180,E1 -11524.662,E2 -11524.662} C_VEL
LIN {X 0,Y 389.473,Z 432.937,A -85,B 0,C 180,E1 -11526.219,E2 -11526.219} C_VEL
LIN {X 0,Y 390.122,Z 427.786,A -85,B 0,C 180,E1 -11527.768,E2 -11527.768} C_VEL
LIN {X 0,Y 390.583,Z 422.224,A -85,B 0,C 180,E1 -11529.062,E2 -11529.062} C_VEL
LIN {X 0,Y 391.194,Z 415.121,A -85,B 0,C 180,E1 -11530.353,E2 -11530.353} C_VEL
LIN {X 0,Y 391.821,Z 408.122,A -85,B 0,C 180,E1 -11531.382,E2 -11531.382} C_VEL
LIN {X 0,Y 392.377,Z 400.721,A -85,B 0,C 180,E1 -11532.283,E2 -11532.283} C_VEL
LIN {X 0,Y 393.033,Z 391.654,A -85,B 0,C 180,E1 -11533.182,E2 -11533.182} C_VEL
LIN {X 0,Y 393.693,Z 380.651,A -85,B 0,C 180,E1 -11534.014,E2 -11534.014} C_VEL
LIN {X 0,Y 394.101,Z 371.717,A -85,B 0,C 180,E1 -11534.526,E2 -11534.526} C_VEL
LIN {X 0,Y 394.427,Z 361.902,A -85,B 0,C 180,E1 -11534.943,E2 -11534.943} C_VEL
LIN {X 0,Y 395.208,Z 337.111,A -85,B 0,C 180,E1 -11535.598,E2 -11535.598} C_VEL
LIN {X 0,Y 396.254,Z 299.725,A -85,B 0,C 180,E1 -11536.581,E2 -11536.581} C_VEL
LIN {X 0,Y 393.127,Z 286.68,A -85,B 0,C 180,E1 -11537.186,E2 -11537.186} C_VEL
LIN {X 0,Y 391.981,Z 282.688,A -85,B 0,C 180,E1 -11537.389,E2 -11537.389} C_VEL
LIN {X 0,Y 391.731,Z 279.113,A -85,B 0,C 180,E1 -11538.344,E2 -11538.344} C_VEL
LIN {X 0,Y 390.094,Z 271.71,A -85,B 0,C 180,E1 -11540.411,E2 -11540.411} C_VEL
LIN {X 0,Y 390.073,Z 271.708,A -85,B 0,C 180,E1 -11543.355,E2 -11543.355} C_VEL
LIN {X 0,Y 390.062,Z 271.712,A -85,B 0,C 180,E1 -11546.775,E2 -11546.775} C_VEL
LIN {X 0,Y 390.046,Z 271.714,A -85,B 0,C 180,E1 -11550.302,E2 -11550.302} C_VEL
LIN {X 0,Y 390.078,Z 271.709,A -85,B 0,C 180,E1 -11554.026,E2 -11554.026} C_VEL
LIN {X 0,Y 390.047,Z 271.711,A -85,B 0,C 180,E1 -11557.782,E2 -11557.782} C_VEL
LIN {X 0,Y 390.028,Z 271.715,A -85,B 0,C 180,E1 -11560.816,E2 -11560.816} C_VEL
LIN {X 0,Y 390.063,Z 271.707,A -85,B 0,C 180,E1 -11563.887,E2 -11563.887} C_VEL
LIN {X 0,Y 390.065,Z 271.709,A -85,B 0,C 180,E1 -11566.79,E2 -11566.79} C_VEL
LIN {X 0,Y 390.042,Z 271.71,A -85,B 0,C 180,E1 -11569.558,E2 -11569.558} C_VEL
LIN {X 0,Y 390.049,Z 271.714,A -85,B 0,C 180,E1 -11572.451,E2 -11572.451} C_VEL
LIN {X 0,Y 390.078,Z 271.704,A -85,B 0,C 180,E1 -11575.976,E2 -11575.976} C_VEL
LIN {X 0,Y 390.056,Z 271.71,A -85,B 0,C 180,E1 -11579.87,E2 -11579.87} C_VEL
LIN {X 0,Y 390.134,Z 271.7,A -85,B 0,C 180,E1 -11583.233,E2 -11583.233} C_VEL
LIN {X 0,Y 390.174,Z 271.811,A -85,B 0,C 180,E1 -11584.292,E2 -11584.292} C_VEL
LIN {X 0,Y 391.659,Z 280.391,A -85,B 0,C 180,E1 -11586.39,E2 -11586.39} C_VEL
LIN {X 0,Y 391.654,Z 285.495,A -85,B 0,C 180,E1 -11587.584,E2 -11587.584} C_VEL
LIN {X 0,Y 390.625,Z 301.995,A -85,B 0,C 180,E1 -11591.376,E2 -11591.376} C_VEL
LIN {X 0,Y 390.292,Z 307.828,A -85,B 0,C 180,E1 -11592.668,E2 -11592.668} C_VEL
LIN {X 0,Y 393.501,Z 327.282,A -85,B 0,C 180,E1 -11593.469,E2 -11593.469} C_VEL
LIN {X 0,Y 394.986,Z 342.93,A -85,B 0,C 180,E1 -11594.017,E2 -11594.017} C_VEL
LIN {X 0,Y 393.5,Z 394.719,A -85,B 0,C 180,E1 -11595.372,E2 -11595.372} C_VEL
LIN {X 0,Y 392.852,Z 406.868,A -85,B 0,C 180,E1 -11595.892,E2 -11595.892} C_VEL
LIN {X 0,Y 392.147,Z 417.178,A -85,B 0,C 180,E1 -11596.527,E2 -11596.527} C_VEL
LIN {X 0,Y 391.494,Z 426.754,A -85,B 0,C 180,E1 -11597.296,E2 -11597.296} C_VEL
LIN {X 0,Y 390.766,Z 436.713,A -85,B 0,C 180,E1 -11598.326,E2 -11598.326} C_VEL
LIN {X 0,Y 390.173,Z 444.594,A -85,B 0,C 180,E1 -11599.36,E2 -11599.36} C_VEL
LIN {X 0,Y 389.71,Z 451.132,A -85,B 0,C 180,E1 -11600.397,E2 -11600.397} C_VEL
LIN {X 0,Y 389.371,Z 456.569,A -85,B 0,C 180,E1 -11601.436,E2 -11601.436} C_VEL
LIN {X 0,Y 389.127,Z 461.092,A -85,B 0,C 180,E1 -11602.476,E2 -11602.476} C_VEL
LIN {X 0,Y 388.842,Z 465.673,A -85,B 0,C 180,E1 -11603.774,E2 -11603.774} C_VEL
LIN {X 0,Y 388.751,Z 471.069,A -85,B 0,C 180,E1 -11605.853,E2 -11605.853} C_VEL
LIN {X 0,Y 388.724,Z 473.05,A -85,B 0,C 180,E1 -11606.891,E2 -11606.891} C_VEL
LIN {X 0,Y 388.8,Z 474.565,A -85,B 0,C 180,E1 -11607.928,E2 -11607.928} C_VEL
LIN {X 0,Y 388.765,Z 475.519,A -85,B 0,C 180,E1 -11608.964,E2 -11608.964} C_VEL
LIN {X 0,Y 388.751,Z 475.896,A -85,B 0,C 180,E1 -11610,E2 -11610} C_VEL
LIN {X 0,Y 388.756,Z 475.805,A -85,B 0,C 180,E1 -11611.036,E2 -11611.036} C_VEL
LIN {X 0,Y 388.761,Z 475.252,A -85,B 0,C 180,E1 -11612.072,E2 -11612.072} C_VEL
LIN {X 0,Y 388.69,Z 474.213,A -85,B 0,C 180,E1 -11613.109,E2 -11613.109} C_VEL
LIN {X 0,Y 388.791,Z 471.552,A -85,B 0,C 180,E1 -11614.666,E2 -11614.666} C_VEL
LIN {X 0,Y 388.841,Z 467.632,A -85,B 0,C 180,E1 -11616.226,E2 -11616.226} C_VEL
LIN {X 0,Y 389.091,Z 464.267,A -85,B 0,C 180,E1 -11617.264,E2 -11617.264} C_VEL
LIN {X 0,Y 389.393,Z 459.02,A -85,B 0,C 180,E1 -11618.563,E2 -11618.563} C_VEL
LIN {X 0,Y 389.834,Z 453.898,A -85,B 0,C 180,E1 -11619.599,E2 -11619.599} C_VEL
LIN {X 0,Y 390.327,Z 447.75,A -85,B 0,C 180,E1 -11620.635,E2 -11620.635} C_VEL
LIN {X 0,Y 390.861,Z 441.308,A -85,B 0,C 180,E1 -11621.539,E2 -11621.539} C_VEL
LIN {X 0,Y 391.449,Z 433.528,A -85,B 0,C 180,E1 -11622.441,E2 -11622.441} C_VEL
LIN {X 0,Y 392.106,Z 425.344,A -85,B 0,C 180,E1 -11623.21,E2 -11623.21} C_VEL
LIN {X 0,Y 392.706,Z 416.836,A -85,B 0,C 180,E1 -11623.849,E2 -11623.849} C_VEL
LIN {X 0,Y 393.279,Z 406.892,A -85,B 0,C 180,E1 -11624.422,E2 -11624.422} C_VEL
LIN {X 0,Y 393.87,Z 394.279,A -85,B 0,C 180,E1 -11624.896,E2 -11624.896} C_VEL
LIN {X 0,Y 394.26,Z 371.936,A -85,B 0,C 180,E1 -11625.346,E2 -11625.346} C_VEL
LIN {X 0,Y 394.439,Z 341.551,A -85,B 0,C 180,E1 -11625.917,E2 -11625.917} C_VEL
LIN {X 0,Y 392.14,Z 324.021,A -85,B 0,C 180,E1 -11626.369,E2 -11626.369} C_VEL
LIN {X 0,Y 390.555,Z 314.545,A -85,B 0,C 180,E1 -11626.654,E2 -11626.654} C_VEL
LIN {X 0,Y 391.595,Z 297.949,A -85,B 0,C 180,E1 -11630.485,E2 -11630.485} C_VEL
LIN {X 0,Y 392.466,Z 286.357,A -85,B 0,C 180,E1 -11633.201,E2 -11633.201} C_VEL
LIN {X 0,Y 391.838,Z 280.547,A -85,B 0,C 180,E1 -11634.646,E2 -11634.646} C_VEL
LIN {X 0,Y 390.162,Z 271.702,A -85,B 0,C 180,E1 -11636.981,E2 -11636.981} C_VEL
LIN {X 0,Y 390.046,Z 271.71,A -85,B 0,C 180,E1 -11640.299,E2 -11640.299} C_VEL
LIN {X 0,Y 390.077,Z 271.709,A -85,B 0,C 180,E1 -11644.024,E2 -11644.024} C_VEL
LIN {X 0,Y 390.047,Z 271.713,A -85,B 0,C 180,E1 -11647.779,E2 -11647.779} C_VEL
LIN {X 0,Y 390.055,Z 271.71,A -85,B 0,C 180,E1 -11650.818,E2 -11650.818} C_VEL
LIN {X 0,Y 390.061,Z 271.706,A -85,B 0,C 180,E1 -11653.885,E2 -11653.885} C_VEL
LIN {X 0,Y 390.063,Z 271.707,A -85,B 0,C 180,E1 -11656.788,E2 -11656.788} C_VEL
LIN {X 0,Y 390.021,Z 271.716,A -85,B 0,C 180,E1 -11659.554,E2 -11659.554} C_VEL
LIN {X 0,Y 390.047,Z 271.708,A -85,B 0,C 180,E1 -11662.448,E2 -11662.448} C_VEL
LIN {X 0,Y 390.076,Z 271.708,A -85,B 0,C 180,E1 -11665.974,E2 -11665.974} C_VEL
LIN {X 0,Y 390.051,Z 271.709,A -85,B 0,C 180,E1 -11669.868,E2 -11669.868} C_VEL
LIN {X 0,Y 390.061,Z 271.706,A -85,B 0,C 180,E1 -11673.225,E2 -11673.225} C_VEL
LIN {X 0,Y 390.073,Z 271.705,A -85,B 0,C 180,E1 -11676.762,E2 -11676.762} C_VEL
LIN {X 0,Y 390.109,Z 271.703,A -85,B 0,C 180,E1 -11679.981,E2 -11679.981} C_VEL
LIN {X 0,Y 390.143,Z 271.693,A -85,B 0,C 180,E1 -11683.246,E2 -11683.246} C_VEL
LIN {X 0,Y 390.199,Z 271.688,A -85,B 0,C 180,E1 -11686.559,E2 -11686.559} C_VEL
LIN {X 0,Y 390.208,Z 271.685,A -85,B 0,C 180,E1 -11690.668,E2 -11690.668} C_VEL
LIN {X 0,Y 390.327,Z 271.67,A -85,B 0,C 180,E1 -11693.795,E2 -11693.795} C_VEL
LIN {X 0,Y 390.414,Z 271.665,A -85,B 0,C 180,E1 -11697.934,E2 -11697.934} C_VEL
LIN {X 0,Y 390.544,Z 271.641,A -85,B 0,C 180,E1 -11699.997,E2 -11699.997} C_VEL
LIN {X 0,Y 390.302,Z 271.674,A -85,B 0,C 180,E1 -11703.093,E2 -11703.093} C_VEL
LIN {X 0,Y 390.272,Z 271.676,A -85,B 0,C 180,E1 -11706.51,E2 -11706.51} C_VEL
LIN {X 0,Y 390.189,Z 271.688,A -85,B 0,C 180,E1 -11709.325,E2 -11709.325} C_VEL
LIN {X 0,Y 390.165,Z 271.698,A -85,B 0,C 180,E1 -11712.479,E2 -11712.479} C_VEL
LIN {X 0,Y 390.132,Z 271.694,A -85,B 0,C 180,E1 -11715.673,E2 -11715.673} C_VEL
LIN {X 0,Y 390.096,Z 271.702,A -85,B 0,C 180,E1 -11718.918,E2 -11718.918} C_VEL
LIN {X 0,Y 390.03,Z 271.714,A -85,B 0,C 180,E1 -11722.23,E2 -11722.23} C_VEL
LIN {X 0,Y 390.107,Z 271.7,A -85,B 0,C 180,E1 -11725.74,E2 -11725.74} C_VEL
LIN {X 0,Y 390.044,Z 271.71,A -85,B 0,C 180,E1 -11729.106,E2 -11729.106} C_VEL
LIN {X 0,Y 390.026,Z 271.717,A -85,B 0,C 180,E1 -11732.718,E2 -11732.718} C_VEL
LIN {X 0,Y 390.037,Z 271.701,A -85,B 0,C 180,E1 -11735.822,E2 -11735.822} C_VEL
LIN {X 0,Y 390.048,Z 271.708,A -85,B 0,C 180,E1 -11739.215,E2 -11739.215} C_VEL
LIN {X 0,Y 390.097,Z 271.708,A -85,B 0,C 180,E1 -11742.383,E2 -11742.383} C_VEL
LIN {X 0,Y 390.095,Z 271.706,A -85,B 0,C 180,E1 -11745.362,E2 -11745.362} C_VEL
LIN {X 0,Y 390.08,Z 271.708,A -85,B 0,C 180,E1 -11748.193,E2 -11748.193} C_VEL
LIN {X 0,Y 390.069,Z 271.71,A -85,B 0,C 180,E1 -11750.905,E2 -11750.905} C_VEL
LIN {X 0,Y 390.055,Z 271.867,A -85,B 0,C 180,E1 -11753.83,E2 -11753.83} C_VEL
LIN {X 0,Y 391.23,Z 278.559,A -85,B 0,C 180,E1 -11755.715,E2 -11755.715} C_VEL
LIN {X 0,Y 391.19,Z 281.239,A -85,B 0,C 180,E1 -11756.425,E2 -11756.425} C_VEL
LIN {X 0,Y 394.994,Z 298.561,A -85,B 0,C 180,E1 -11756.97,E2 -11756.97} C_VEL
LIN {X 0,Y 394.281,Z 357.432,A -85,B 0,C 180,E1 -11758.088,E2 -11758.088} C_VEL
LIN {X 0,Y 394.049,Z 367.114,A -85,B 0,C 180,E1 -11758.405,E2 -11758.405} C_VEL
LIN {X 0,Y 393.676,Z 377.332,A -85,B 0,C 180,E1 -11758.903,E2 -11758.903} C_VEL
LIN {X 0,Y 393.101,Z 388.628,A -85,B 0,C 180,E1 -11759.683,E2 -11759.683} C_VEL
LIN {X 0,Y 392.46,Z 397.524,A -85,B 0,C 180,E1 -11760.498,E2 -11760.498} C_VEL
LIN {X 0,Y 391.866,Z 405.044,A -85,B 0,C 180,E1 -11761.35,E2 -11761.35} C_VEL
LIN {X 0,Y 391.352,Z 411.066,A -85,B 0,C 180,E1 -11762.166,E2 -11762.166} C_VEL
LIN {X 0,Y 390.764,Z 417.841,A -85,B 0,C 180,E1 -11763.28,E2 -11763.28} C_VEL
LIN {X 0,Y 390.313,Z 423.392,A -85,B 0,C 180,E1 -11764.396,E2 -11764.396} C_VEL
LIN {X 0,Y 389.902,Z 427.937,A -85,B 0,C 180,E1 -11765.508,E2 -11765.508} C_VEL
LIN {X 0,Y 389.531,Z 431.635,A -85,B 0,C 180,E1 -11766.614,E2 -11766.614} C_VEL
LIN {X 0,Y 389.16,Z 435.806,A -85,B 0,C 180,E1 -11768.271,E2 -11768.271} C_VEL
LIN {X 0,Y 388.843,Z 438.696,A -85,B 0,C 180,E1 -11770.012,E2 -11770.012} C_VEL
LIN {X 0,Y 388.726,Z 439.615,A -85,B 0,C 180,E1 -11771.008,E2 -11771.008} C_VEL
LIN {X 0,Y 388.662,Z 440.107,A -85,B 0,C 180,E1 -11772.097,E2 -11772.097} C_VEL
LIN {X 0,Y 388.675,Z 440.014,A -85,B 0,C 180,E1 -11773.385,E2 -11773.385} C_VEL
LIN {X 0,Y 388.687,Z 439.543,A -85,B 0,C 180,E1 -11774.263,E2 -11774.263} C_VEL
LIN {X 0,Y 388.729,Z 438.485,A -85,B 0,C 180,E1 -11775.338,E2 -11775.338} C_VEL
LIN {X 0,Y 388.862,Z 436.811,A -85,B 0,C 180,E1 -11776.411,E2 -11776.411} C_VEL
LIN {X 0,Y 389.058,Z 433.236,A -85,B 0,C 180,E1 -11778.01,E2 -11778.01} C_VEL
LIN {X 0,Y 389.237,Z 430.093,A -85,B 0,C 180,E1 -11779.072,E2 -11779.072} C_VEL
LIN {X 0,Y 389.533,Z 425.102,A -85,B 0,C 180,E1 -11780.393,E2 -11780.393} C_VEL
LIN {X 0,Y 389.95,Z 418.773,A -85,B 0,C 180,E1 -11781.71,E2 -11781.71} C_VEL
LIN {X 0,Y 390.327,Z 412.584,A -85,B 0,C 180,E1 -11782.759,E2 -11782.759} C_VEL
LIN {X 0,Y 390.677,Z 406.095,A -85,B 0,C 180,E1 -11783.674,E2 -11783.674} C_VEL
LIN {X 0,Y 391.097,Z 399.447,A -85,B 0,C 180,E1 -11784.457,E2 -11784.457} C_VEL
LIN {X 0,Y 391.555,Z 391.386,A -85,B 0,C 180,E1 -11785.238,E2 -11785.238} C_VEL
LIN {X 0,Y 391.898,Z 383.079,A -85,B 0,C 180,E1 -11785.887,E2 -11785.887} C_VEL
LIN {X 0,Y 392.167,Z 374.648,A -85,B 0,C 180,E1 -11786.404,E2 -11786.404} C_VEL
LIN {X 0,Y 392.45,Z 365.437,A -85,B 0,C 180,E1 -11786.824,E2 -11786.824} C_VEL
LIN {X 0,Y 392.644,Z 355.957,A -85,B 0,C 180,E1 -11787.115,E2 -11787.115} C_VEL
LIN {X 0,Y 393.133,Z 297.251,A -85,B 0,C 180,E1 -11788.207,E2 -11788.207} C_VEL
LIN {X 0,Y 390.35,Z 281.038,A -85,B 0,C 180,E1 -11788.614,E2 -11788.614} C_VEL
LIN {X 0,Y 390.591,Z 276.013,A -85,B 0,C 180,E1 -11789.956,E2 -11789.956} C_VEL
LIN {X 0,Y 390.337,Z 274.426,A -85,B 0,C 180,E1 -11790.476,E2 -11790.476} C_VEL
LIN {X 0,Y 389.494,Z 273.358,A -85,B 0,C 180,E1 -11791.014,E2 -11791.014} C_VEL
LIN {X 0,Y 386.899,Z 272.409,A -85,B 0,C 180,E1 -11792.113,E2 -11792.113} C_VEL
LIN {X 0,Y 384.234,Z 272.438,A -85,B 0,C 180,E1 -11793.262,E2 -11793.262} C_VEL
LIN {X 0,Y 383.124,Z 272.571,A -85,B 0,C 180,E1 -11794.156,E2 -11794.156} C_VEL
LIN {X 0,Y 383.056,Z 272.579,A -85,B 0,C 180,E1 -11794.459,E2 -11794.459} C_VEL
LIN {X 0,Y 383.247,Z 272.555,A -85,B 0,C 180,E1 -11796.317,E2 -11796.317} C_VEL
LIN {X 0,Y 383.187,Z 272.563,A -85,B 0,C 180,E1 -11798.438,E2 -11798.438} C_VEL
LIN {X 0,Y 383.062,Z 272.581,A -85,B 0,C 180,E1 -11801.643,E2 -11801.643} C_VEL
LIN {X 0,Y 383.075,Z 272.579,A -85,B 0,C 180,E1 -11804.883,E2 -11804.883} C_VEL
LIN {X 0,Y 383.029,Z 272.582,A -85,B 0,C 180,E1 -11808.175,E2 -11808.175} C_VEL
LIN {X 0,Y 382.966,Z 272.595,A -85,B 0,C 180,E1 -11811.533,E2 -11811.533} C_VEL
LIN {X 0,Y 382.986,Z 272.589,A -85,B 0,C 180,E1 -11814.965,E2 -11814.965} C_VEL
LIN {X 0,Y 382.955,Z 272.591,A -85,B 0,C 180,E1 -11818.5,E2 -11818.5} C_VEL
LIN {X 0,Y 382.98,Z 272.589,A -85,B 0,C 180,E1 -11822.153,E2 -11822.153} C_VEL
LIN {X 0,Y 382.99,Z 272.587,A -85,B 0,C 180,E1 -11824.671,E2 -11824.671} C_VEL
LIN {X 0,Y 382.967,Z 272.593,A -85,B 0,C 180,E1 -11827.906,E2 -11827.906} C_VEL
LIN {X 0,Y 382.938,Z 272.597,A -85,B 0,C 180,E1 -11831.354,E2 -11831.354} C_VEL
LIN {X 0,Y 382.972,Z 272.59,A -85,B 0,C 180,E1 -11834.307,E2 -11834.307} C_VEL
LIN {X 0,Y 382.99,Z 272.589,A -85,B 0,C 180,E1 -11837.244,E2 -11837.244} C_VEL
LIN {X 0,Y 382.994,Z 272.588,A -85,B 0,C 180,E1 -11840.418,E2 -11840.418} C_VEL
LIN {X 0,Y 383.008,Z 272.589,A -85,B 0,C 180,E1 -11844.048,E2 -11844.048} C_VEL
LIN {X 0,Y 382.972,Z 272.593,A -85,B 0,C 180,E1 -11847.582,E2 -11847.582} C_VEL
LIN {X 0,Y 382.967,Z 272.593,A -85,B 0,C 180,E1 -11850.303,E2 -11850.303} C_VEL
LIN {X 0,Y 382.993,Z 272.592,A -85,B 0,C 180,E1 -11854.048,E2 -11854.048} C_VEL
LIN {X 0,Y 382.982,Z 272.589,A -85,B 0,C 180,E1 -11857.338,E2 -11857.338} C_VEL
LIN {X 0,Y 383.056,Z 272.58,A -85,B 0,C 180,E1 -11860.72,E2 -11860.72} C_VEL
LIN {X 0,Y 383.173,Z 272.687,A -85,B 0,C 180,E1 -11862.668,E2 -11862.668} C_VEL
LIN {X 0,Y 383.078,Z 280.388,A -85,B 0,C 180,E1 -11864.645,E2 -11864.645} C_VEL
LIN {X 0,Y 385.631,Z 298.483,A -85,B 0,C 180,E1 -11865.162,E2 -11865.162} C_VEL
LIN {X 0,Y 384.635,Z 359.162,A -85,B 0,C 180,E1 -11866.633,E2 -11866.633} C_VEL
LIN {X 0,Y 384.438,Z 368.344,A -85,B 0,C 180,E1 -11866.996,E2 -11866.996} C_VEL
LIN {X 0,Y 384.137,Z 378.025,A -85,B 0,C 180,E1 -11867.523,E2 -11867.523} C_VEL
LIN {X 0,Y 383.827,Z 388.204,A -85,B 0,C 180,E1 -11868.25,E2 -11868.25} C_VEL
LIN {X 0,Y 383.402,Z 398.047,A -85,B 0,C 180,E1 -11869.174,E2 -11869.174} C_VEL
LIN {X 0,Y 383.082,Z 405.949,A -85,B 0,C 180,E1 -11870.1,E2 -11870.1} C_VEL
LIN {X 0,Y 382.631,Z 414.226,A -85,B 0,C 180,E1 -11871.288,E2 -11871.288} C_VEL
LIN {X 0,Y 382.375,Z 421.622,A -85,B 0,C 180,E1 -11872.612,E2 -11872.612} C_VEL
LIN {X 0,Y 382.112,Z 426.371,A -85,B 0,C 180,E1 -11873.668,E2 -11873.668} C_VEL
LIN {X 0,Y 382.016,Z 430.306,A -85,B 0,C 180,E1 -11874.726,E2 -11874.726} C_VEL
LIN {X 0,Y 381.836,Z 434.812,A -85,B 0,C 180,E1 -11876.31,E2 -11876.31} C_VEL
LIN {X 0,Y 381.726,Z 437.958,A -85,B 0,C 180,E1 -11877.893,E2 -11877.893} C_VEL
LIN {X 0,Y 381.701,Z 439.338,A -85,B 0,C 180,E1 -11878.948,E2 -11878.948} C_VEL
LIN {X 0,Y 381.682,Z 440.192,A -85,B 0,C 180,E1 -11880.003,E2 -11880.003} C_VEL
LIN {X 0,Y 381.723,Z 440.523,A -85,B 0,C 180,E1 -11881.058,E2 -11881.058} C_VEL
LIN {X 0,Y 381.83,Z 440.266,A -85,B 0,C 180,E1 -11882.113,E2 -11882.113} C_VEL
LIN {X 0,Y 382.014,Z 439.415,A -85,B 0,C 180,E1 -11883.167,E2 -11883.167} C_VEL
LIN {X 0,Y 382.264,Z 438.028,A -85,B 0,C 180,E1 -11884.221,E2 -11884.221} C_VEL
LIN {X 0,Y 382.462,Z 434.98,A -85,B 0,C 180,E1 -11885.804,E2 -11885.804} C_VEL
LIN {X 0,Y 382.946,Z 430.451,A -85,B 0,C 180,E1 -11887.384,E2 -11887.384} C_VEL
LIN {X 0,Y 383.387,Z 425.448,A -85,B 0,C 180,E1 -11888.702,E2 -11888.702} C_VEL
LIN {X 0,Y 384.065,Z 419.142,A -85,B 0,C 180,E1 -11890.014,E2 -11890.014} C_VEL
LIN {X 0,Y 384.825,Z 411.266,A -85,B 0,C 180,E1 -11891.325,E2 -11891.325} C_VEL
LIN {X 0,Y 385.574,Z 402.095,A -85,B 0,C 180,E1 -11892.504,E2 -11892.504} C_VEL
LIN {X 0,Y 386.239,Z 393.217,A -85,B 0,C 180,E1 -11893.418,E2 -11893.418} C_VEL
LIN {X 0,Y 387.011,Z 381.847,A -85,B 0,C 180,E1 -11894.328,E2 -11894.328} C_VEL
LIN {X 0,Y 387.508,Z 371.965,A -85,B 0,C 180,E1 -11894.913,E2 -11894.913} C_VEL
LIN {X 0,Y 387.865,Z 362.268,A -85,B 0,C 180,E1 -11895.336,E2 -11895.336} C_VEL
LIN {X 0,Y 388.785,Z 334.906,A -85,B 0,C 180,E1 -11896.082,E2 -11896.082} C_VEL
LIN {X 0,Y 389.814,Z 300.849,A -85,B 0,C 180,E1 -11897.005,E2 -11897.005} C_VEL
LIN {X 0,Y 386.938,Z 288.933,A -85,B 0,C 180,E1 -11897.591,E2 -11897.591} C_VEL
LIN {X 0,Y 385.179,Z 282.918,A -85,B 0,C 180,E1 -11897.958,E2 -11897.958} C_VEL
LIN {X 0,Y 383.747,Z 275.332,A -85,B 0,C 180,E1 -11900.086,E2 -11900.086} C_VEL
LIN {X 0,Y 383.044,Z 272.586,A -85,B 0,C 180,E1 -11900.95,E2 -11900.95} C_VEL
LIN {X 0,Y 383.021,Z 272.589,A -85,B 0,C 180,E1 -11903.811,E2 -11903.811} C_VEL
LIN {X 0,Y 383.002,Z 272.59,A -85,B 0,C 180,E1 -11907.309,E2 -11907.309} C_VEL
LIN {X 0,Y 382.991,Z 272.592,A -85,B 0,C 180,E1 -11910.92,E2 -11910.92} C_VEL
LIN {X 0,Y 383.021,Z 272.589,A -85,B 0,C 180,E1 -11914.67,E2 -11914.67} C_VEL
LIN {X 0,Y 383.003,Z 272.589,A -85,B 0,C 180,E1 -11917.904,E2 -11917.904} C_VEL
LIN {X 0,Y 382.972,Z 272.592,A -85,B 0,C 180,E1 -11921.352,E2 -11921.352} C_VEL
LIN {X 0,Y 383.005,Z 272.589,A -85,B 0,C 180,E1 -11924.304,E2 -11924.304} C_VEL
LIN {X 0,Y 383.021,Z 272.584,A -85,B 0,C 180,E1 -11927.241,E2 -11927.241} C_VEL
LIN {X 0,Y 383.003,Z 272.589,A -85,B 0,C 180,E1 -11930.419,E2 -11930.419} C_VEL
LIN {X 0,Y 383.031,Z 272.581,A -85,B 0,C 180,E1 -11934.045,E2 -11934.045} C_VEL
LIN {X 0,Y 382.994,Z 272.589,A -85,B 0,C 180,E1 -11937.579,E2 -11937.579} C_VEL
LIN {X 0,Y 383.001,Z 272.589,A -85,B 0,C 180,E1 -11940.301,E2 -11940.301} C_VEL
LIN {X 0,Y 383.162,Z 272.694,A -85,B 0,C 180,E1 -11944.153,E2 -11944.153} C_VEL
LIN {X 0,Y 384.748,Z 282.501,A -85,B 0,C 180,E1 -11946.59,E2 -11946.59} C_VEL
LIN {X 0,Y 384.251,Z 292.224,A -85,B 0,C 180,E1 -11948.879,E2 -11948.879} C_VEL
LIN {X 0,Y 383.351,Z 306.095,A -85,B 0,C 180,E1 -11952.082,E2 -11952.082} C_VEL
LIN {X 0,Y 386.814,Z 326.603,A -85,B 0,C 180,E1 -11952.982,E2 -11952.982} C_VEL
LIN {X 0,Y 388.202,Z 339.961,A -85,B 0,C 180,E1 -11953.485,E2 -11953.485} C_VEL
LIN {X 0,Y 388.383,Z 345.713,A -85,B 0,C 180,E1 -11953.665,E2 -11953.665} C_VEL
LIN {X 0,Y 386.882,Z 394.788,A -85,B 0,C 180,E1 -11954.998,E2 -11954.998} C_VEL
LIN {X 0,Y 386.208,Z 406.32,A -85,B 0,C 180,E1 -11955.51,E2 -11955.51} C_VEL
LIN {X 0,Y 385.441,Z 416.587,A -85,B 0,C 180,E1 -11956.154,E2 -11956.154} C_VEL
LIN {X 0,Y 384.744,Z 426.209,A -85,B 0,C 180,E1 -11956.935,E2 -11956.935} C_VEL
LIN {X 0,Y 383.97,Z 436.224,A -85,B 0,C 180,E1 -11957.983,E2 -11957.983} C_VEL
LIN {X 0,Y 383.427,Z 443.261,A -85,B 0,C 180,E1 -11958.903,E2 -11958.903} C_VEL
LIN {X 0,Y 382.782,Z 449.943,A -85,B 0,C 180,E1 -11959.955,E2 -11959.955} C_VEL
LIN {X 0,Y 382.341,Z 456.727,A -85,B 0,C 180,E1 -11961.277,E2 -11961.277} C_VEL
LIN {X 0,Y 382.032,Z 462.159,A -85,B 0,C 180,E1 -11962.601,E2 -11962.601} C_VEL
LIN {X 0,Y 381.691,Z 467.247,A -85,B 0,C 180,E1 -11964.22,E2 -11964.22} C_VEL
LIN {X 0,Y 381.682,Z 470.656,A -85,B 0,C 180,E1 -11965.776,E2 -11965.776} C_VEL
LIN {X 0,Y 381.63,Z 472.644,A -85,B 0,C 180,E1 -11966.833,E2 -11966.833} C_VEL
LIN {X 0,Y 381.7,Z 474.189,A -85,B 0,C 180,E1 -11967.889,E2 -11967.889} C_VEL
LIN {X 0,Y 381.696,Z 475.15,A -85,B 0,C 180,E1 -11968.945,E2 -11968.945} C_VEL
LIN {X 0,Y 381.681,Z 475.554,A -85,B 0,C 180,E1 -11970,E2 -11970} C_VEL
LIN {X 0,Y 381.687,Z 475.494,A -85,B 0,C 180,E1 -11971.055,E2 -11971.055} C_VEL
LIN {X 0,Y 381.659,Z 474.97,A -85,B 0,C 180,E1 -11972.11,E2 -11972.11} C_VEL
LIN {X 0,Y 381.599,Z 473.95,A -85,B 0,C 180,E1 -11973.167,E2 -11973.167} C_VEL
LIN {X 0,Y 381.702,Z 471.338,A -85,B 0,C 180,E1 -11974.753,E2 -11974.753} C_VEL
LIN {X 0,Y 381.764,Z 467.824,A -85,B 0,C 180,E1 -11976.215,E2 -11976.215} C_VEL
LIN {X 0,Y 382.042,Z 464.138,A -85,B 0,C 180,E1 -11977.398,E2 -11977.398} C_VEL
LIN {X 0,Y 382.363,Z 458.942,A -85,B 0,C 180,E1 -11978.722,E2 -11978.722} C_VEL
LIN {X 0,Y 382.902,Z 452.453,A -85,B 0,C 180,E1 -11980.042,E2 -11980.042} C_VEL
LIN {X 0,Y 383.657,Z 444.374,A -85,B 0,C 180,E1 -11981.357,E2 -11981.357} C_VEL
LIN {X 0,Y 384.434,Z 434.957,A -85,B 0,C 180,E1 -11982.538,E2 -11982.538} C_VEL
LIN {X 0,Y 385.132,Z 427.156,A -85,B 0,C 180,E1 -11983.32,E2 -11983.32} C_VEL
LIN {X 0,Y 385.725,Z 419.175,A -85,B 0,C 180,E1 -11983.97,E2 -11983.97} C_VEL
LIN {X 0,Y 386.29,Z 410.009,A -85,B 0,C 180,E1 -11984.554,E2 -11984.554} C_VEL
LIN {X 0,Y 386.806,Z 400.376,A -85,B 0,C 180,E1 -11985.004,E2 -11985.004} C_VEL
LIN {X 0,Y 387.171,Z 391.474,A -85,B 0,C 180,E1 -11985.284,E2 -11985.284} C_VEL
LIN {X 0,Y 387.766,Z 342.572,A -85,B 0,C 180,E1 -11986.231,E2 -11986.231} C_VEL
LIN {X 0,Y 385.507,Z 325.301,A -85,B 0,C 180,E1 -11986.687,E2 -11986.687} C_VEL
LIN {X 0,Y 383.591,Z 314.24,A -85,B 0,C 180,E1 -11987.02,E2 -11987.02} C_VEL
LIN {X 0,Y 384.69,Z 298.051,A -85,B 0,C 180,E1 -11990.832,E2 -11990.832} C_VEL
LIN {X 0,Y 385.539,Z 287.463,A -85,B 0,C 180,E1 -11993.358,E2 -11993.358} C_VEL
LIN {X 0,Y 384.872,Z 281.668,A -85,B 0,C 180,E1 -11994.834,E2 -11994.834} C_VEL
LIN {X 0,Y 383.143,Z 272.574,A -85,B 0,C 180,E1 -11997.295,E2 -11997.295} C_VEL
LIN {X 0,Y 382.99,Z 272.592,A -85,B 0,C 180,E1 -12000.918,E2 -12000.918} C_VEL
LIN {X 0,Y 383.019,Z 272.588,A -85,B 0,C 180,E1 -12004.668,E2 -12004.668} C_VEL
LIN {X 0,Y 383.003,Z 272.589,A -85,B 0,C 180,E1 -12007.901,E2 -12007.901} C_VEL
LIN {X 0,Y 382.985,Z 272.591,A -85,B 0,C 180,E1 -12011.347,E2 -12011.347} C_VEL
LIN {X 0,Y 383.003,Z 272.584,A -85,B 0,C 180,E1 -12014.302,E2 -12014.302} C_VEL
LIN {X 0,Y 383.018,Z 272.585,A -85,B 0,C 180,E1 -12017.239,E2 -12017.239} C_VEL
LIN {X 0,Y 382.994,Z 272.584,A -85,B 0,C 180,E1 -12020.417,E2 -12020.417} C_VEL
LIN {X 0,Y 383.032,Z 272.58,A -85,B 0,C 180,E1 -12024.043,E2 -12024.043} C_VEL
LIN {X 0,Y 382.994,Z 272.591,A -85,B 0,C 180,E1 -12027.576,E2 -12027.576} C_VEL
LIN {X 0,Y 382.987,Z 272.589,A -85,B 0,C 180,E1 -12030.297,E2 -12030.297} C_VEL
LIN {X 0,Y 383.029,Z 272.582,A -85,B 0,C 180,E1 -12034.036,E2 -12034.036} C_VEL
LIN {X 0,Y 382.998,Z 272.588,A -85,B 0,C 180,E1 -12037.332,E2 -12037.332} C_VEL
LIN {X 0,Y 383.064,Z 272.578,A -85,B 0,C 180,E1 -12040.714,E2 -12040.714} C_VEL
LIN {X 0,Y 383.085,Z 272.572,A -85,B 0,C 180,E1 -12044.024,E2 -12044.024} C_VEL
LIN {X 0,Y 383.14,Z 272.567,A -85,B 0,C 180,E1 -12047.281,E2 -12047.281} C_VEL
LIN {X 0,Y 383.154,Z 272.565,A -85,B 0,C 180,E1 -12050.495,E2 -12050.495} C_VEL
LIN {X 0,Y 383.283,Z 272.548,A -85,B 0,C 180,E1 -12053.68,E2 -12053.68} C_VEL
LIN {X 0,Y 383.38,Z 272.541,A -85,B 0,C 180,E1 -12057.896,E2 -12057.896} C_VEL
LIN {X 0,Y 383.514,Z 272.516,A -85,B 0,C 180,E1 -12059.997,E2 -12059.997} C_VEL
LIN {X 0,Y 383.238,Z 272.554,A -85,B 0,C 180,E1 -12063.15,E2 -12063.15} C_VEL
LIN {X 0,Y 383.235,Z 272.554,A -85,B 0,C 180,E1 -12066.498,E2 -12066.498} C_VEL
LIN {X 0,Y 383.139,Z 272.567,A -85,B 0,C 180,E1 -12069.499,E2 -12069.499} C_VEL
LIN {X 0,Y 383.119,Z 272.572,A -85,B 0,C 180,E1 -12073.532,E2 -12073.532} C_VEL
LIN {X 0,Y 383.086,Z 272.575,A -85,B 0,C 180,E1 -12077.451,E2 -12077.451} C_VEL
LIN {X 0,Y 383.019,Z 272.583,A -85,B 0,C 180,E1 -12080.643,E2 -12080.643} C_VEL
LIN {X 0,Y 383.022,Z 272.584,A -85,B 0,C 180,E1 -12083.803,E2 -12083.803} C_VEL
LIN {X 0,Y 383.067,Z 272.58,A -85,B 0,C 180,E1 -12086.119,E2 -12086.119} C_VEL
LIN {X 0,Y 382.977,Z 272.59,A -85,B 0,C 180,E1 -12089.696,E2 -12089.696} C_VEL
LIN {X 0,Y 382.986,Z 272.589,A -85,B 0,C 180,E1 -12093.397,E2 -12093.397} C_VEL
LIN {X 0,Y 383.013,Z 272.576,A -85,B 0,C 180,E1 -12096.161,E2 -12096.161} C_VEL
LIN {X 0,Y 382.994,Z 272.586,A -85,B 0,C 180,E1 -12099.954,E2 -12099.954} C_VEL
LIN {X 0,Y 383.043,Z 272.586,A -85,B 0,C 180,E1 -12102.785,E2 -12102.785} C_VEL
LIN {X 0,Y 383.048,Z 272.583,A -85,B 0,C 180,E1 -12105.797,E2 -12105.797} C_VEL
LIN {X 0,Y 383.019,Z 272.587,A -85,B 0,C 180,E1 -12108.783,E2 -12108.783} C_VEL
LIN {X 0,Y 382.976,Z 272.596,A -85,B 0,C 180,E1 -12112.093,E2 -12112.093} C_VEL
LIN {X 0,Y 383.018,Z 272.743,A -85,B 0,C 180,E1 -12113.55,E2 -12113.55} C_VEL
LIN {X 0,Y 384.279,Z 279.4,A -85,B 0,C 180,E1 -12115.462,E2 -12115.462} C_VEL
LIN {X 0,Y 384.344,Z 281.831,A -85,B 0,C 180,E1 -12116.072,E2 -12116.072} C_VEL
LIN {X 0,Y 388.319,Z 299.509,A -85,B 0,C 180,E1 -12116.64,E2 -12116.64} C_VEL
LIN {X 0,Y 387.531,Z 358.086,A -85,B 0,C 180,E1 -12117.772,E2 -12117.772} C_VEL
LIN {X 0,Y 387.299,Z 367.665,A -85,B 0,C 180,E1 -12118.095,E2 -12118.095} C_VEL
LIN {X 0,Y 386.905,Z 377.982,A -85,B 0,C 180,E1 -12118.611,E2 -12118.611} C_VEL
LIN {X 0,Y 386.307,Z 388.858,A -85,B 0,C 180,E1 -12119.376,E2 -12119.376} C_VEL
LIN {X 0,Y 385.638,Z 397.938,A -85,B 0,C 180,E1 -12120.224,E2 -12120.224} C_VEL
LIN {X 0,Y 384.985,Z 405.698,A -85,B 0,C 180,E1 -12121.123,E2 -12121.123} C_VEL
LIN {X 0,Y 384.471,Z 411.453,A -85,B 0,C 180,E1 -12121.92,E2 -12121.92} C_VEL
LIN {X 0,Y 383.843,Z 418.219,A -85,B 0,C 180,E1 -12123.054,E2 -12123.054} C_VEL
LIN {X 0,Y 383.327,Z 423.756,A -85,B 0,C 180,E1 -12124.187,E2 -12124.187} C_VEL
LIN {X 0,Y 382.914,Z 428.298,A -85,B 0,C 180,E1 -12125.32,E2 -12125.32} C_VEL
LIN {X 0,Y 382.396,Z 432.879,A -85,B 0,C 180,E1 -12126.758,E2 -12126.758} C_VEL
LIN {X 0,Y 382.175,Z 435.552,A -85,B 0,C 180,E1 -12127.853,E2 -12127.853} C_VEL
LIN {X 0,Y 382.061,Z 436.754,A -85,B 0,C 180,E1 -12128.414,E2 -12128.414} C_VEL
LIN {X 0,Y 381.779,Z 438.961,A -85,B 0,C 180,E1 -12129.841,E2 -12129.841} C_VEL
LIN {X 0,Y 381.595,Z 440.359,A -85,B 0,C 180,E1 -12131.754,E2 -12131.754} C_VEL
LIN {X 0,Y 381.566,Z 440.364,A -85,B 0,C 180,E1 -12133.272,E2 -12133.272} C_VEL
LIN {X 0,Y 381.584,Z 440.104,A -85,B 0,C 180,E1 -12133.963,E2 -12133.963} C_VEL
LIN {X 0,Y 381.613,Z 439.107,A -85,B 0,C 180,E1 -12135.059,E2 -12135.059} C_VEL
LIN {X 0,Y 381.799,Z 436.631,A -85,B 0,C 180,E1 -12136.698,E2 -12136.698} C_VEL
LIN {X 0,Y 382.016,Z 432.762,A -85,B 0,C 180,E1 -12138.325,E2 -12138.325} C_VEL
LIN {X 0,Y 382.359,Z 427.48,A -85,B 0,C 180,E1 -12139.944,E2 -12139.944} C_VEL
LIN {X 0,Y 382.741,Z 420.51,A -85,B 0,C 180,E1 -12141.553,E2 -12141.553} C_VEL
LIN {X 0,Y 383.158,Z 414.585,A -85,B 0,C 180,E1 -12142.623,E2 -12142.623} C_VEL
LIN {X 0,Y 383.615,Z 407.372,A -85,B 0,C 180,E1 -12143.689,E2 -12143.689} C_VEL
LIN {X 0,Y 384.105,Z 399.676,A -85,B 0,C 180,E1 -12144.62,E2 -12144.62} C_VEL
LIN {X 0,Y 384.57,Z 391.597,A -85,B 0,C 180,E1 -12145.414,E2 -12145.414} C_VEL
LIN {X 0,Y 384.922,Z 383.265,A -85,B 0,C 180,E1 -12146.074,E2 -12146.074} C_VEL
LIN {X 0,Y 385.196,Z 374.799,A -85,B 0,C 180,E1 -12146.601,E2 -12146.601} C_VEL
LIN {X 0,Y 385.505,Z 364.697,A -85,B 0,C 180,E1 -12147.061,E2 -12147.061} C_VEL
LIN {X 0,Y 385.712,Z 353.299,A -85,B 0,C 180,E1 -12147.389,E2 -12147.389} C_VEL
LIN {X 0,Y 386.212,Z 298.096,A -85,B 0,C 180,E1 -12148.42,E2 -12148.42} C_VEL
LIN {X 0,Y 383.371,Z 281.314,A -85,B 0,C 180,E1 -12148.851,E2 -12148.851} C_VEL
LIN {X 0,Y 383.573,Z 275.142,A -85,B 0,C 180,E1 -12150.525,E2 -12150.525} C_VEL
LIN {X 0,Y 383.314,Z 272.551,A -85,B 0,C 180,E1 -12151.313,E2 -12151.313} C_VEL
LIN {X 0,Y 383.216,Z 272.565,A -85,B 0,C 180,E1 -12153.154,E2 -12153.154} C_VEL
LIN {X 0,Y 383.056,Z 272.579,A -85,B 0,C 180,E1 -12154.459,E2 -12154.459} C_VEL
LIN {X 0,Y 382.457,Z 272.658,A -85,B 0,C 180,E1 -12155.338,E2 -12155.338} C_VEL
LIN {X 0,Y 379.657,Z 273.004,A -85,B 0,C 180,E1 -12156.769,E2 -12156.769} C_VEL
LIN {X 0,Y 377.238,Z 273.304,A -85,B 0,C 180,E1 -12157.925,E2 -12157.925} C_VEL
LIN {X 0,Y 376.183,Z 273.437,A -85,B 0,C 180,E1 -12158.818,E2 -12158.818} C_VEL
LIN {X 0,Y 376.09,Z 273.446,A -85,B 0,C 180,E1 -12159.121,E2 -12159.121} C_VEL
LIN {X 0,Y 376.069,Z 273.452,A -85,B 0,C 180,E1 -12162.959,E2 -12162.959} C_VEL
LIN {X 0,Y 375.994,Z 273.458,A -85,B 0,C 180,E1 -12166.283,E2 -12166.283} C_VEL
LIN {X 0,Y 375.964,Z 273.465,A -85,B 0,C 180,E1 -12169.663,E2 -12169.663} C_VEL
LIN {X 0,Y 375.946,Z 273.468,A -85,B 0,C 180,E1 -12173.663,E2 -12173.663} C_VEL
LIN {X 0,Y 375.896,Z 273.47,A -85,B 0,C 180,E1 -12176.662,E2 -12176.662} C_VEL
LIN {X 0,Y 375.889,Z 273.474,A -85,B 0,C 180,E1 -12179.086,E2 -12179.086} C_VEL
LIN {X 0,Y 375.928,Z 273.473,A -85,B 0,C 180,E1 -12181.565,E2 -12181.565} C_VEL
LIN {X 0,Y 375.929,Z 273.471,A -85,B 0,C 180,E1 -12185.419,E2 -12185.419} C_VEL
LIN {X 0,Y 375.909,Z 273.47,A -85,B 0,C 180,E1 -12188.266,E2 -12188.266} C_VEL
LIN {X 0,Y 375.895,Z 273.477,A -85,B 0,C 180,E1 -12191.601,E2 -12191.601} C_VEL
LIN {X 0,Y 375.904,Z 273.47,A -85,B 0,C 180,E1 -12194.735,E2 -12194.735} C_VEL
LIN {X 0,Y 375.914,Z 273.469,A -85,B 0,C 180,E1 -12198.403,E2 -12198.403} C_VEL
LIN {X 0,Y 375.953,Z 273.47,A -85,B 0,C 180,E1 -12201.734,E2 -12201.734} C_VEL
LIN {X 0,Y 375.964,Z 273.464,A -85,B 0,C 180,E1 -12205.337,E2 -12205.337} C_VEL
LIN {X 0,Y 375.943,Z 273.466,A -85,B 0,C 180,E1 -12208.442,E2 -12208.442} C_VEL
LIN {X 0,Y 375.923,Z 273.471,A -85,B 0,C 180,E1 -12212.14,E2 -12212.14} C_VEL
LIN {X 0,Y 375.962,Z 273.466,A -85,B 0,C 180,E1 -12215.721,E2 -12215.721} C_VEL
LIN {X 0,Y 375.991,Z 273.459,A -85,B 0,C 180,E1 -12219.202,E2 -12219.202} C_VEL
LIN {X 0,Y 376.147,Z 273.556,A -85,B 0,C 180,E1 -12222.645,E2 -12222.645} C_VEL
LIN {X 0,Y 376.041,Z 280.565,A -85,B 0,C 180,E1 -12224.454,E2 -12224.454} C_VEL
LIN {X 0,Y 378.653,Z 299.474,A -85,B 0,C 180,E1 -12225.021,E2 -12225.021} C_VEL
LIN {X 0,Y 377.578,Z 359.202,A -85,B 0,C 180,E1 -12226.516,E2 -12226.516} C_VEL
LIN {X 0,Y 377.338,Z 369.812,A -85,B 0,C 180,E1 -12226.952,E2 -12226.952} C_VEL
LIN {X 0,Y 377.008,Z 380.295,A -85,B 0,C 180,E1 -12227.557,E2 -12227.557} C_VEL
LIN {X 0,Y 376.661,Z 391.409,A -85,B 0,C 180,E1 -12228.433,E2 -12228.433} C_VEL
LIN {X 0,Y 376.308,Z 399.46,A -85,B 0,C 180,E1 -12229.24,E2 -12229.24} C_VEL
LIN {X 0,Y 375.963,Z 407.195,A -85,B 0,C 180,E1 -12230.183,E2 -12230.183} C_VEL
LIN {X 0,Y 375.504,Z 415.353,A -85,B 0,C 180,E1 -12231.393,E2 -12231.393} C_VEL
LIN {X 0,Y 375.253,Z 422.528,A -85,B 0,C 180,E1 -12232.741,E2 -12232.741} C_VEL
LIN {X 0,Y 374.964,Z 428.171,A -85,B 0,C 180,E1 -12234.087,E2 -12234.087} C_VEL
LIN {X 0,Y 374.888,Z 431.851,A -85,B 0,C 180,E1 -12235.164,E2 -12235.164} C_VEL
LIN {X 0,Y 374.699,Z 436.067,A -85,B 0,C 180,E1 -12236.778,E2 -12236.778} C_VEL
LIN {X 0,Y 374.63,Z 438.092,A -85,B 0,C 180,E1 -12237.853,E2 -12237.853} C_VEL
LIN {X 0,Y 374.616,Z 439.558,A -85,B 0,C 180,E1 -12238.929,E2 -12238.929} C_VEL
LIN {X 0,Y 374.614,Z 440.491,A -85,B 0,C 180,E1 -12240.003,E2 -12240.003} C_VEL
LIN {X 0,Y 374.656,Z 440.878,A -85,B 0,C 180,E1 -12241.078,E2 -12241.078} C_VEL
LIN {X 0,Y 374.77,Z 440.655,A -85,B 0,C 180,E1 -12242.153,E2 -12242.153} C_VEL
LIN {X 0,Y 374.966,Z 439.884,A -85,B 0,C 180,E1 -12243.227,E2 -12243.227} C_VEL
LIN {X 0,Y 375.226,Z 438.586,A -85,B 0,C 180,E1 -12244.3,E2 -12244.3} C_VEL
LIN {X 0,Y 375.438,Z 435.631,A -85,B 0,C 180,E1 -12245.913,E2 -12245.913} C_VEL
LIN {X 0,Y 375.686,Z 432.855,A -85,B 0,C 180,E1 -12246.987,E2 -12246.987} C_VEL
LIN {X 0,Y 376.225,Z 428.553,A -85,B 0,C 180,E1 -12248.3,E2 -12248.3} C_VEL
LIN {X 0,Y 376.977,Z 421.532,A -85,B 0,C 180,E1 -12249.933,E2 -12249.933} C_VEL
LIN {X 0,Y 377.576,Z 415.714,A -85,B 0,C 180,E1 -12251.002,E2 -12251.002} C_VEL
LIN {X 0,Y 378.301,Z 408.717,A -85,B 0,C 180,E1 -12252.067,E2 -12252.067} C_VEL
LIN {X 0,Y 379.075,Z 400.176,A -85,B 0,C 180,E1 -12253.13,E2 -12253.13} C_VEL
LIN {X 0,Y 379.984,Z 389.19,A -85,B 0,C 180,E1 -12254.189,E2 -12254.189} C_VEL
LIN {X 0,Y 380.605,Z 379.293,A -85,B 0,C 180,E1 -12254.916,E2 -12254.916} C_VEL
LIN {X 0,Y 381.139,Z 368.634,A -85,B 0,C 180,E1 -12255.511,E2 -12255.511} C_VEL
LIN {X 0,Y 381.656,Z 355.868,A -85,B 0,C 180,E1 -12255.969,E2 -12255.969} C_VEL
LIN {X 0,Y 383.531,Z 302.385,A -85,B 0,C 180,E1 -12257.442,E2 -12257.442} C_VEL
LIN {X 0,Y 380.197,Z 288.843,A -85,B 0,C 180,E1 -12258.149,E2 -12258.149} C_VEL
LIN {X 0,Y 378.285,Z 283.427,A -85,B 0,C 180,E1 -12258.511,E2 -12258.511} C_VEL
LIN {X 0,Y 376.34,Z 274.952,A -85,B 0,C 180,E1 -12260.975,E2 -12260.975} C_VEL
LIN {X 0,Y 375.966,Z 273.468,A -85,B 0,C 180,E1 -12261.452,E2 -12261.452} C_VEL
LIN {X 0,Y 375.97,Z 273.468,A -85,B 0,C 180,E1 -12264.286,E2 -12264.286} C_VEL
LIN {X 0,Y 375.943,Z 273.469,A -85,B 0,C 180,E1 -12267.866,E2 -12267.866} C_VEL
LIN {X 0,Y 375.966,Z 273.466,A -85,B 0,C 180,E1 -12271.564,E2 -12271.564} C_VEL
LIN {X 0,Y 375.959,Z 273.465,A -85,B 0,C 180,E1 -12275.418,E2 -12275.418} C_VEL
LIN {X 0,Y 375.945,Z 273.469,A -85,B 0,C 180,E1 -12278.264,E2 -12278.264} C_VEL
LIN {X 0,Y 375.928,Z 273.469,A -85,B 0,C 180,E1 -12281.599,E2 -12281.599} C_VEL
LIN {X 0,Y 375.936,Z 273.468,A -85,B 0,C 180,E1 -12284.732,E2 -12284.732} C_VEL
LIN {X 0,Y 375.939,Z 273.47,A -85,B 0,C 180,E1 -12288.401,E2 -12288.401} C_VEL
LIN {X 0,Y 375.947,Z 273.466,A -85,B 0,C 180,E1 -12291.738,E2 -12291.738} C_VEL
LIN {X 0,Y 375.988,Z 273.461,A -85,B 0,C 180,E1 -12295.334,E2 -12295.334} C_VEL
LIN {X 0,Y 375.966,Z 273.463,A -85,B 0,C 180,E1 -12298.439,E2 -12298.439} C_VEL
LIN {X 0,Y 375.995,Z 273.463,A -85,B 0,C 180,E1 -12302.141,E2 -12302.141} C_VEL
LIN {X 0,Y 376.078,Z 273.469,A -85,B 0,C 180,E1 -12303.979,E2 -12303.979} C_VEL
LIN {X 0,Y 377.68,Z 283.07,A -85,B 0,C 180,E1 -12306.417,E2 -12306.417} C_VEL
LIN {X 0,Y 377.49,Z 289.021,A -85,B 0,C 180,E1 -12307.851,E2 -12307.851} C_VEL
LIN {X 0,Y 376.438,Z 304.056,A -85,B 0,C 180,E1 -12311.424,E2 -12311.424} C_VEL
LIN {X 0,Y 380.308,Z 326.269,A -85,B 0,C 180,E1 -12312.479,E2 -12312.479} C_VEL
LIN {X 0,Y 381.832,Z 341.575,A -85,B 0,C 180,E1 -12313.077,E2 -12313.077} C_VEL
LIN {X 0,Y 381.901,Z 349.577,A -85,B 0,C 180,E1 -12313.329,E2 -12313.329} C_VEL
LIN {X 0,Y 380.304,Z 394.71,A -85,B 0,C 180,E1 -12314.594,E2 -12314.594} C_VEL
LIN {X 0,Y 379.587,Z 406.097,A -85,B 0,C 180,E1 -12315.114,E2 -12315.114} C_VEL
LIN {X 0,Y 378.79,Z 416.314,A -85,B 0,C 180,E1 -12315.768,E2 -12315.768} C_VEL
LIN {X 0,Y 378.022,Z 425.844,A -85,B 0,C 180,E1 -12316.562,E2 -12316.562} C_VEL
LIN {X 0,Y 377.142,Z 435.801,A -85,B 0,C 180,E1 -12317.625,E2 -12317.625} C_VEL
LIN {X 0,Y 376.493,Z 443.683,A -85,B 0,C 180,E1 -12318.696,E2 -12318.696} C_VEL
LIN {X 0,Y 375.801,Z 450.252,A -85,B 0,C 180,E1 -12319.766,E2 -12319.766} C_VEL
LIN {X 0,Y 375.405,Z 455.709,A -85,B 0,C 180,E1 -12320.843,E2 -12320.843} C_VEL
LIN {X 0,Y 375.02,Z 461.273,A -85,B 0,C 180,E1 -12322.191,E2 -12322.191} C_VEL
LIN {X 0,Y 374.688,Z 466.397,A -85,B 0,C 180,E1 -12323.795,E2 -12323.795} C_VEL
LIN {X 0,Y 374.625,Z 469.533,A -85,B 0,C 180,E1 -12325.157,E2 -12325.157} C_VEL
LIN {X 0,Y 374.601,Z 473.802,A -85,B 0,C 180,E1 -12327.849,E2 -12327.849} C_VEL
LIN {X 0,Y 374.629,Z 474.771,A -85,B 0,C 180,E1 -12328.925,E2 -12328.925} C_VEL
LIN {X 0,Y 374.612,Z 475.21,A -85,B 0,C 180,E1 -12330,E2 -12330} C_VEL
LIN {X 0,Y 374.62,Z 475.184,A -85,B 0,C 180,E1 -12331.075,E2 -12331.075} C_VEL
LIN {X 0,Y 374.558,Z 474.693,A -85,B 0,C 180,E1 -12332.15,E2 -12332.15} C_VEL
LIN {X 0,Y 374.512,Z 473.688,A -85,B 0,C 180,E1 -12333.227,E2 -12333.227} C_VEL
LIN {X 0,Y 374.614,Z 471.133,A -85,B 0,C 180,E1 -12334.843,E2 -12334.843} C_VEL
LIN {X 0,Y 374.725,Z 467.294,A -85,B 0,C 180,E1 -12336.461,E2 -12336.461} C_VEL
LIN {X 0,Y 375.112,Z 462.087,A -85,B 0,C 180,E1 -12338.078,E2 -12338.078} C_VEL
LIN {X 0,Y 375.695,Z 455.263,A -85,B 0,C 180,E1 -12339.692,E2 -12339.692} C_VEL
LIN {X 0,Y 376.362,Z 447.825,A -85,B 0,C 180,E1 -12341.035,E2 -12341.035} C_VEL
LIN {X 0,Y 377.059,Z 440.508,A -85,B 0,C 180,E1 -12342.104,E2 -12342.104} C_VEL
LIN {X 0,Y 377.746,Z 432.699,A -85,B 0,C 180,E1 -12343.037,E2 -12343.037} C_VEL
LIN {X 0,Y 378.436,Z 424.482,A -85,B 0,C 180,E1 -12343.833,E2 -12343.833} C_VEL
LIN {X 0,Y 379.256,Z 414.072,A -85,B 0,C 180,E1 -12344.624,E2 -12344.624} C_VEL
LIN {X 0,Y 379.905,Z 402.63,A -85,B 0,C 180,E1 -12345.237,E2 -12345.237} C_VEL
LIN {X 0,Y 380.421,Z 392.599,A -85,B 0,C 180,E1 -12345.585,E2 -12345.585} C_VEL
LIN {X 0,Y 380.888,Z 363.076,A -85,B 0,C 180,E1 -12346.184,E2 -12346.184} C_VEL
LIN {X 0,Y 380.99,Z 342.066,A -85,B 0,C 180,E1 -12346.597,E2 -12346.597} C_VEL
LIN {X 0,Y 378.446,Z 323.955,A -85,B 0,C 180,E1 -12347.099,E2 -12347.099} C_VEL
LIN {X 0,Y 376.66,Z 313.842,A -85,B 0,C 180,E1 -12347.421,E2 -12347.421} C_VEL
LIN {X 0,Y 377.655,Z 300.159,A -85,B 0,C 180,E1 -12350.706,E2 -12350.706} C_VEL
LIN {X 0,Y 378.603,Z 288.585,A -85,B 0,C 180,E1 -12353.522,E2 -12353.522} C_VEL
LIN {X 0,Y 378.055,Z 283.671,A -85,B 0,C 180,E1 -12354.798,E2 -12354.798} C_VEL
LIN {X 0,Y 376.069,Z 273.452,A -85,B 0,C 180,E1 -12357.626,E2 -12357.626} C_VEL
LIN {X 0,Y 375.964,Z 273.464,A -85,B 0,C 180,E1 -12361.561,E2 -12361.561} C_VEL
LIN {X 0,Y 375.957,Z 273.46,A -85,B 0,C 180,E1 -12365.415,E2 -12365.415} C_VEL
LIN {X 0,Y 375.946,Z 273.467,A -85,B 0,C 180,E1 -12368.262,E2 -12368.262} C_VEL
LIN {X 0,Y 375.937,Z 273.468,A -85,B 0,C 180,E1 -12371.598,E2 -12371.598} C_VEL
LIN {X 0,Y 375.934,Z 273.468,A -85,B 0,C 180,E1 -12375.267,E2 -12375.267} C_VEL
LIN {X 0,Y 375.928,Z 273.467,A -85,B 0,C 180,E1 -12378.4,E2 -12378.4} C_VEL
LIN {X 0,Y 375.961,Z 273.466,A -85,B 0,C 180,E1 -12381.908,E2 -12381.908} C_VEL
LIN {X 0,Y 375.987,Z 273.457,A -85,B 0,C 180,E1 -12385.331,E2 -12385.331} C_VEL
LIN {X 0,Y 375.964,Z 273.458,A -85,B 0,C 180,E1 -12388.436,E2 -12388.436} C_VEL
LIN {X 0,Y 375.941,Z 273.465,A -85,B 0,C 180,E1 -12392.134,E2 -12392.134} C_VEL
LIN {X 0,Y 375.984,Z 273.465,A -85,B 0,C 180,E1 -12395.715,E2 -12395.715} C_VEL
LIN {X 0,Y 376.004,Z 273.451,A -85,B 0,C 180,E1 -12399.195,E2 -12399.195} C_VEL
LIN {X 0,Y 376.038,Z 273.449,A -85,B 0,C 180,E1 -12402.597,E2 -12402.597} C_VEL
LIN {X 0,Y 376.094,Z 273.446,A -85,B 0,C 180,E1 -12406.34,E2 -12406.34} C_VEL
LIN {X 0,Y 376.122,Z 273.442,A -85,B 0,C 180,E1 -12410.316,E2 -12410.316} C_VEL
LIN {X 0,Y 376.241,Z 273.425,A -85,B 0,C 180,E1 -12413.562,E2 -12413.562} C_VEL
LIN {X 0,Y 376.345,Z 273.416,A -85,B 0,C 180,E1 -12417.856,E2 -12417.856} C_VEL
LIN {X 0,Y 376.483,Z 273.391,A -85,B 0,C 180,E1 -12419.997,E2 -12419.997} C_VEL
LIN {X 0,Y 376.349,Z 273.417,A -85,B 0,C 180,E1 -12422.137,E2 -12422.137} C_VEL
LIN {X 0,Y 376.205,Z 273.432,A -85,B 0,C 180,E1 -12426.483,E2 -12426.483} C_VEL
LIN {X 0,Y 376.109,Z 273.444,A -85,B 0,C 180,E1 -12429.678,E2 -12429.678} C_VEL
LIN {X 0,Y 376.083,Z 273.449,A -85,B 0,C 180,E1 -12433.654,E2 -12433.654} C_VEL
LIN {X 0,Y 376.036,Z 273.454,A -85,B 0,C 180,E1 -12437.603,E2 -12437.603} C_VEL
LIN {X 0,Y 375.968,Z 273.462,A -85,B 0,C 180,E1 -12440.828,E2 -12440.828} C_VEL
LIN {X 0,Y 375.982,Z 273.461,A -85,B 0,C 180,E1 -12444.278,E2 -12444.278} C_VEL
LIN {X 0,Y 376.007,Z 273.462,A -85,B 0,C 180,E1 -12446.648,E2 -12446.648} C_VEL
LIN {X 0,Y 375.949,Z 273.47,A -85,B 0,C 180,E1 -12450.309,E2 -12450.309} C_VEL
LIN {X 0,Y 375.943,Z 273.469,A -85,B 0,C 180,E1 -12454.108,E2 -12454.108} C_VEL
LIN {X 0,Y 375.934,Z 273.462,A -85,B 0,C 180,E1 -12456.738,E2 -12456.738} C_VEL
LIN {X 0,Y 375.973,Z 273.46,A -85,B 0,C 180,E1 -12459.968,E2 -12459.968} C_VEL
LIN {X 0,Y 375.976,Z 273.46,A -85,B 0,C 180,E1 -12463.752,E2 -12463.752} C_VEL
LIN {X 0,Y 375.975,Z 273.462,A -85,B 0,C 180,E1 -12466.797,E2 -12466.797} C_VEL
LIN {X 0,Y 375.973,Z 273.466,A -85,B 0,C 180,E1 -12470.024,E2 -12470.024} C_VEL
LIN {X 0,Y 375.939,Z 273.527,A -85,B 0,C 180,E1 -12473.216,E2 -12473.216} C_VEL
LIN {X 0,Y 377.371,Z 280.91,A -85,B 0,C 180,E1 -12475.387,E2 -12475.387} C_VEL
LIN {X 0,Y 377.405,Z 281.995,A -85,B 0,C 180,E1 -12475.675,E2 -12475.675} C_VEL
LIN {X 0,Y 381.611,Z 300.337,A -85,B 0,C 180,E1 -12476.285,E2 -12476.285} C_VEL
LIN {X 0,Y 380.835,Z 358.072,A -85,B 0,C 180,E1 -12477.423,E2 -12477.423} C_VEL
LIN {X 0,Y 380.608,Z 367.688,A -85,B 0,C 180,E1 -12477.749,E2 -12477.749} C_VEL
LIN {X 0,Y 380.204,Z 377.4,A -85,B 0,C 180,E1 -12478.234,E2 -12478.234} C_VEL
LIN {X 0,Y 379.589,Z 387.618,A -85,B 0,C 180,E1 -12478.929,E2 -12478.929} C_VEL
LIN {X 0,Y 378.93,Z 397.066,A -85,B 0,C 180,E1 -12479.796,E2 -12479.796} C_VEL
LIN {X 0,Y 378.237,Z 405.204,A -85,B 0,C 180,E1 -12480.735,E2 -12480.735} C_VEL
LIN {X 0,Y 377.584,Z 411.848,A -85,B 0,C 180,E1 -12481.665,E2 -12481.665} C_VEL
LIN {X 0,Y 376.903,Z 418.593,A -85,B 0,C 180,E1 -12482.817,E2 -12482.817} C_VEL
LIN {X 0,Y 376.46,Z 423.113,A -85,B 0,C 180,E1 -12483.737,E2 -12483.737} C_VEL
LIN {X 0,Y 375.992,Z 427.643,A -85,B 0,C 180,E1 -12484.834,E2 -12484.834} C_VEL
LIN {X 0,Y 375.529,Z 432.074,A -85,B 0,C 180,E1 -12486.175,E2 -12486.175} C_VEL
LIN {X 0,Y 375.194,Z 435.298,A -85,B 0,C 180,E1 -12487.419,E2 -12487.419} C_VEL
LIN {X 0,Y 374.827,Z 438.436,A -85,B 0,C 180,E1 -12489.13,E2 -12489.13} C_VEL
LIN {X 0,Y 374.636,Z 439.795,A -85,B 0,C 180,E1 -12490.265,E2 -12490.265} C_VEL
LIN {X 0,Y 374.525,Z 440.613,A -85,B 0,C 180,E1 -12491.397,E2 -12491.397} C_VEL
LIN {X 0,Y 374.485,Z 440.892,A -85,B 0,C 180,E1 -12492.526,E2 -12492.526} C_VEL
LIN {X 0,Y 374.491,Z 440.557,A -85,B 0,C 180,E1 -12493.65,E2 -12493.65} C_VEL
LIN {X 0,Y 374.5,Z 439.68,A -85,B 0,C 180,E1 -12494.768,E2 -12494.768} C_VEL
LIN {X 0,Y 374.618,Z 438.28,A -85,B 0,C 180,E1 -12495.884,E2 -12495.884} C_VEL
LIN {X 0,Y 374.858,Z 434.96,A -85,B 0,C 180,E1 -12497.639,E2 -12497.639} C_VEL
LIN {X 0,Y 375.086,Z 430.687,A -85,B 0,C 180,E1 -12499.201,E2 -12499.201} C_VEL
LIN {X 0,Y 375.426,Z 425.669,A -85,B 0,C 180,E1 -12500.573,E2 -12500.573} C_VEL
LIN {X 0,Y 375.87,Z 419.226,A -85,B 0,C 180,E1 -12501.957,E2 -12501.957} C_VEL
LIN {X 0,Y 376.246,Z 413.114,A -85,B 0,C 180,E1 -12503.026,E2 -12503.026} C_VEL
LIN {X 0,Y 376.666,Z 406.586,A -85,B 0,C 180,E1 -12503.976,E2 -12503.976} C_VEL
LIN {X 0,Y 377.095,Z 399.912,A -85,B 0,C 180,E1 -12504.787,E2 -12504.787} C_VEL
LIN {X 0,Y 377.572,Z 391.816,A -85,B 0,C 180,E1 -12505.597,E2 -12505.597} C_VEL
LIN {X 0,Y 377.949,Z 383.452,A -85,B 0,C 180,E1 -12506.269,E2 -12506.269} C_VEL
LIN {X 0,Y 378.252,Z 374.935,A -85,B 0,C 180,E1 -12506.805,E2 -12506.805} C_VEL
LIN {X 0,Y 378.571,Z 364.766,A -85,B 0,C 180,E1 -12507.274,E2 -12507.274} C_VEL
LIN {X 0,Y 378.768,Z 353.143,A -85,B 0,C 180,E1 -12507.607,E2 -12507.607} C_VEL
LIN {X 0,Y 379.371,Z 299.442,A -85,B 0,C 180,E1 -12508.624,E2 -12508.624} C_VEL
LIN {X 0,Y 376.375,Z 281.582,A -85,B 0,C 180,E1 -12509.097,E2 -12509.097} C_VEL
LIN {X 0,Y 376.57,Z 276.342,A -85,B 0,C 180,E1 -12510.535,E2 -12510.535} C_VEL
LIN {X 0,Y 376.291,Z 273.425,A -85,B 0,C 180,E1 -12511.405,E2 -12511.405} C_VEL
LIN {X 0,Y 376.134,Z 273.446,A -85,B 0,C 180,E1 -12515.361,E2 -12515.361} C_VEL
LIN {X 0,Y 376.185,Z 273.435,A -85,B 0,C 180,E1 -12518.083,E2 -12518.083} C_VEL
LIN {X 0,Y 376.09,Z 273.446,A -85,B 0,C 180,E1 -12519.121,E2 -12519.121} C_VEL
LIN {X 0,Y 375.408,Z 273.533,A -85,B 0,C 180,E1 -12520.015,E2 -12520.015} C_VEL
LIN {X 0,Y 372.564,Z 273.891,A -85,B 0,C 180,E1 -12521.468,E2 -12521.468} C_VEL
LIN {X 0,Y 370.151,Z 274.192,A -85,B 0,C 180,E1 -12522.642,E2 -12522.642} C_VEL
LIN {X 0,Y 369.095,Z 274.322,A -85,B 0,C 180,E1 -12523.551,E2 -12523.551} C_VEL
LIN {X 0,Y 368.997,Z 274.331,A -85,B 0,C 180,E1 -12523.858,E2 -12523.858} C_VEL
LIN {X 0,Y 368.968,Z 274.336,A -85,B 0,C 180,E1 -12527.77,E2 -12527.77} C_VEL
LIN {X 0,Y 368.897,Z 274.347,A -85,B 0,C 180,E1 -12531.222,E2 -12531.222} C_VEL
LIN {X 0,Y 368.895,Z 274.343,A -85,B 0,C 180,E1 -12534.78,E2 -12534.78} C_VEL
LIN {X 0,Y 368.885,Z 274.344,A -85,B 0,C 180,E1 -12538.444,E2 -12538.444} C_VEL
LIN {X 0,Y 368.869,Z 274.346,A -85,B 0,C 180,E1 -12542.241,E2 -12542.241} C_VEL
LIN {X 0,Y 368.901,Z 274.343,A -85,B 0,C 180,E1 -12545.004,E2 -12545.004} C_VEL
LIN {X 0,Y 368.851,Z 274.348,A -85,B 0,C 180,E1 -12548.637,E2 -12548.637} C_VEL
LIN {X 0,Y 368.847,Z 274.352,A -85,B 0,C 180,E1 -12552.011,E2 -12552.011} C_VEL
LIN {X 0,Y 368.857,Z 274.349,A -85,B 0,C 180,E1 -12555.179,E2 -12555.179} C_VEL
LIN {X 0,Y 368.863,Z 274.349,A -85,B 0,C 180,E1 -12558.181,E2 -12558.181} C_VEL
LIN {X 0,Y 368.887,Z 274.346,A -85,B 0,C 180,E1 -12561.364,E2 -12561.364} C_VEL
LIN {X 0,Y 368.92,Z 274.34,A -85,B 0,C 180,E1 -12565.15,E2 -12565.15} C_VEL
LIN {X 0,Y 368.899,Z 274.342,A -85,B 0,C 180,E1 -12569.049,E2 -12569.049} C_VEL
LIN {X 0,Y 368.904,Z 274.344,A -85,B 0,C 180,E1 -12571.563,E2 -12571.563} C_VEL
LIN {X 0,Y 368.916,Z 274.341,A -85,B 0,C 180,E1 -12575.226,E2 -12575.226} C_VEL
LIN {X 0,Y 368.912,Z 274.341,A -85,B 0,C 180,E1 -12578.985,E2 -12578.985} C_VEL
LIN {X 0,Y 369.083,Z 274.445,A -85,B 0,C 180,E1 -12582.624,E2 -12582.624} C_VEL
LIN {X 0,Y 369.016,Z 280.858,A -85,B 0,C 180,E1 -12584.292,E2 -12584.292} C_VEL
LIN {X 0,Y 371.625,Z 300.289,A -85,B 0,C 180,E1 -12584.879,E2 -12584.879} C_VEL
LIN {X 0,Y 370.548,Z 359.256,A -85,B 0,C 180,E1 -12586.395,E2 -12586.395} C_VEL
LIN {X 0,Y 370.304,Z 369.902,A -85,B 0,C 180,E1 -12586.84,E2 -12586.84} C_VEL
LIN {X 0,Y 369.961,Z 380.423,A -85,B 0,C 180,E1 -12587.455,E2 -12587.455} C_VEL
LIN {X 0,Y 369.6,Z 391.598,A -85,B 0,C 180,E1 -12588.348,E2 -12588.348} C_VEL
LIN {X 0,Y 369.241,Z 399.678,A -85,B 0,C 180,E1 -12589.17,E2 -12589.17} C_VEL
LIN {X 0,Y 368.883,Z 407.443,A -85,B 0,C 180,E1 -12590.131,E2 -12590.131} C_VEL
LIN {X 0,Y 368.462,Z 414.766,A -85,B 0,C 180,E1 -12591.227,E2 -12591.227} C_VEL
LIN {X 0,Y 368.188,Z 422.338,A -85,B 0,C 180,E1 -12592.629,E2 -12592.629} C_VEL
LIN {X 0,Y 367.877,Z 427.998,A -85,B 0,C 180,E1 -12593.972,E2 -12593.972} C_VEL
LIN {X 0,Y 367.735,Z 433.365,A -85,B 0,C 180,E1 -12595.619,E2 -12595.619} C_VEL
LIN {X 0,Y 367.573,Z 437.291,A -85,B 0,C 180,E1 -12597.264,E2 -12597.264} C_VEL
LIN {X 0,Y 367.533,Z 439.761,A -85,B 0,C 180,E1 -12598.908,E2 -12598.908} C_VEL
LIN {X 0,Y 367.547,Z 440.779,A -85,B 0,C 180,E1 -12600.004,E2 -12600.004} C_VEL
LIN {X 0,Y 367.592,Z 441.207,A -85,B 0,C 180,E1 -12601.099,E2 -12601.099} C_VEL
LIN {X 0,Y 367.713,Z 441.047,A -85,B 0,C 180,E1 -12602.194,E2 -12602.194} C_VEL
LIN {X 0,Y 367.921,Z 440.365,A -85,B 0,C 180,E1 -12603.289,E2 -12603.289} C_VEL
LIN {X 0,Y 368.191,Z 439.154,A -85,B 0,C 180,E1 -12604.382,E2 -12604.382} C_VEL
LIN {X 0,Y 368.418,Z 436.282,A -85,B 0,C 180,E1 -12606.026,E2 -12606.026} C_VEL
LIN {X 0,Y 368.688,Z 433.59,A -85,B 0,C 180,E1 -12607.121,E2 -12607.121} C_VEL
LIN {X 0,Y 369.27,Z 429.402,A -85,B 0,C 180,E1 -12608.458,E2 -12608.458} C_VEL
LIN {X 0,Y 369.964,Z 423.888,A -85,B 0,C 180,E1 -12609.847,E2 -12609.847} C_VEL
LIN {X 0,Y 370.734,Z 416.999,A -85,B 0,C 180,E1 -12611.207,E2 -12611.207} C_VEL
LIN {X 0,Y 371.494,Z 410.155,A -85,B 0,C 180,E1 -12612.291,E2 -12612.291} C_VEL
LIN {X 0,Y 372.316,Z 401.787,A -85,B 0,C 180,E1 -12613.373,E2 -12613.373} C_VEL
LIN {X 0,Y 373.123,Z 392.755,A -85,B 0,C 180,E1 -12614.316,E2 -12614.316} C_VEL
LIN {X 0,Y 373.916,Z 381.847,A -85,B 0,C 180,E1 -12615.19,E2 -12615.19} C_VEL
LIN {X 0,Y 374.508,Z 371.912,A -85,B 0,C 180,E1 -12615.793,E2 -12615.793} C_VEL
LIN {X 0,Y 375.019,Z 361.286,A -85,B 0,C 180,E1 -12616.259,E2 -12616.259} C_VEL
LIN {X 0,Y 377.182,Z 303.393,A -85,B 0,C 180,E1 -12617.928,E2 -12617.928} C_VEL
LIN {X 0,Y 373.866,Z 290.269,A -85,B 0,C 180,E1 -12618.663,E2 -12618.663} C_VEL
LIN {X 0,Y 371.23,Z 283.712,A -85,B 0,C 180,E1 -12619.172,E2 -12619.172} C_VEL
LIN {X 0,Y 369.554,Z 276.772,A -85,B 0,C 180,E1 -12621.273,E2 -12621.273} C_VEL
LIN {X 0,Y 368.928,Z 274.344,A -85,B 0,C 180,E1 -12622.03,E2 -12622.03} C_VEL
LIN {X 0,Y 368.909,Z 274.346,A -85,B 0,C 180,E1 -12624.782,E2 -12624.782} C_VEL
LIN {X 0,Y 368.925,Z 274.342,A -85,B 0,C 180,E1 -12628.443,E2 -12628.443} C_VEL
LIN {X 0,Y 368.907,Z 274.347,A -85,B 0,C 180,E1 -12632.24,E2 -12632.24} C_VEL
LIN {X 0,Y 368.933,Z 274.342,A -85,B 0,C 180,E1 -12635.002,E2 -12635.002} C_VEL
LIN {X 0,Y 368.886,Z 274.349,A -85,B 0,C 180,E1 -12638.635,E2 -12638.635} C_VEL
LIN {X 0,Y 368.881,Z 274.347,A -85,B 0,C 180,E1 -12642.009,E2 -12642.009} C_VEL
LIN {X 0,Y 368.889,Z 274.345,A -85,B 0,C 180,E1 -12645.177,E2 -12645.177} C_VEL
LIN {X 0,Y 368.888,Z 274.346,A -85,B 0,C 180,E1 -12648.178,E2 -12648.178} C_VEL
LIN {X 0,Y 368.889,Z 274.346,A -85,B 0,C 180,E1 -12651.367,E2 -12651.367} C_VEL
LIN {X 0,Y 368.945,Z 274.339,A -85,B 0,C 180,E1 -12655.147,E2 -12655.147} C_VEL
LIN {X 0,Y 368.923,Z 274.342,A -85,B 0,C 180,E1 -12659.046,E2 -12659.046} C_VEL
LIN {X 0,Y 368.978,Z 274.334,A -85,B 0,C 180,E1 -12662.797,E2 -12662.797} C_VEL
LIN {X 0,Y 369.036,Z 274.384,A -85,B 0,C 180,E1 -12663.84,E2 -12663.84} C_VEL
LIN {X 0,Y 370.574,Z 283.103,A -85,B 0,C 180,E1 -12666.101,E2 -12666.101} C_VEL
LIN {X 0,Y 370.646,Z 287.227,A -85,B 0,C 180,E1 -12667.125,E2 -12667.125} C_VEL
LIN {X 0,Y 369.636,Z 302.171,A -85,B 0,C 180,E1 -12670.753,E2 -12670.753} C_VEL
LIN {X 0,Y 374.103,Z 328.262,A -85,B 0,C 180,E1 -12672.045,E2 -12672.045} C_VEL
LIN {X 0,Y 375.452,Z 342.16,A -85,B 0,C 180,E1 -12672.614,E2 -12672.614} C_VEL
LIN {X 0,Y 375.445,Z 351.203,A -85,B 0,C 180,E1 -12672.901,E2 -12672.901} C_VEL
LIN {X 0,Y 373.825,Z 394.044,A -85,B 0,C 180,E1 -12674.146,E2 -12674.146} C_VEL
LIN {X 0,Y 373.012,Z 405.975,A -85,B 0,C 180,E1 -12674.705,E2 -12674.705} C_VEL
LIN {X 0,Y 372.167,Z 416.047,A -85,B 0,C 180,E1 -12675.37,E2 -12675.37} C_VEL
LIN {X 0,Y 371.325,Z 425.568,A -85,B 0,C 180,E1 -12676.175,E2 -12676.175} C_VEL
LIN {X 0,Y 370.36,Z 435.505,A -85,B 0,C 180,E1 -12677.256,E2 -12677.256} C_VEL
LIN {X 0,Y 369.685,Z 442.513,A -85,B 0,C 180,E1 -12678.207,E2 -12678.207} C_VEL
LIN {X 0,Y 369.013,Z 449.175,A -85,B 0,C 180,E1 -12679.298,E2 -12679.298} C_VEL
LIN {X 0,Y 368.406,Z 455.952,A -85,B 0,C 180,E1 -12680.668,E2 -12680.668} C_VEL
LIN {X 0,Y 367.98,Z 461.399,A -85,B 0,C 180,E1 -12682.041,E2 -12682.041} C_VEL
LIN {X 0,Y 367.583,Z 466.768,A -85,B 0,C 180,E1 -12683.846,E2 -12683.846} C_VEL
LIN {X 0,Y 367.52,Z 470.316,A -85,B 0,C 180,E1 -12685.613,E2 -12685.613} C_VEL
LIN {X 0,Y 367.502,Z 473.407,A -85,B 0,C 180,E1 -12687.808,E2 -12687.808} C_VEL
LIN {X 0,Y 367.563,Z 474.391,A -85,B 0,C 180,E1 -12688.904,E2 -12688.904} C_VEL
LIN {X 0,Y 367.546,Z 474.865,A -85,B 0,C 180,E1 -12690,E2 -12690} C_VEL
LIN {X 0,Y 367.535,Z 474.874,A -85,B 0,C 180,E1 -12691.095,E2 -12691.095} C_VEL
LIN {X 0,Y 367.457,Z 474.417,A -85,B 0,C 180,E1 -12692.192,E2 -12692.192} C_VEL
LIN {X 0,Y 367.429,Z 473.419,A -85,B 0,C 180,E1 -12693.289,E2 -12693.289} C_VEL
LIN {X 0,Y 367.527,Z 470.928,A -85,B 0,C 180,E1 -12694.936,E2 -12694.936} C_VEL
LIN {X 0,Y 367.658,Z 467.128,A -85,B 0,C 180,E1 -12696.586,E2 -12696.586} C_VEL
LIN {X 0,Y 368.063,Z 461.967,A -85,B 0,C 180,E1 -12698.233,E2 -12698.233} C_VEL
LIN {X 0,Y 368.556,Z 456.44,A -85,B 0,C 180,E1 -12699.605,E2 -12699.605} C_VEL
LIN {X 0,Y 369.232,Z 449.552,A -85,B 0,C 180,E1 -12700.972,E2 -12700.972} C_VEL
LIN {X 0,Y 370.128,Z 440.66,A -85,B 0,C 180,E1 -12702.334,E2 -12702.334} C_VEL
LIN {X 0,Y 370.857,Z 432.959,A -85,B 0,C 180,E1 -12703.284,E2 -12703.284} C_VEL
LIN {X 0,Y 371.569,Z 424.881,A -85,B 0,C 180,E1 -12704.094,E2 -12704.094} C_VEL
LIN {X 0,Y 372.303,Z 416.512,A -85,B 0,C 180,E1 -12704.764,E2 -12704.764} C_VEL
LIN {X 0,Y 372.867,Z 407.982,A -85,B 0,C 180,E1 -12705.3,E2 -12705.3} C_VEL
LIN {X 0,Y 373.424,Z 399.444,A -85,B 0,C 180,E1 -12705.697,E2 -12705.697} C_VEL
LIN {X 0,Y 373.786,Z 389.553,A -85,B 0,C 180,E1 -12706.012,E2 -12706.012} C_VEL
LIN {X 0,Y 374.371,Z 343.487,A -85,B 0,C 180,E1 -12706.933,E2 -12706.933} C_VEL
LIN {X 0,Y 371.982,Z 325.909,A -85,B 0,C 180,E1 -12707.427,E2 -12707.427} C_VEL
LIN {X 0,Y 369.745,Z 313.484,A -85,B 0,C 180,E1 -12707.837,E2 -12707.837} C_VEL
LIN {X 0,Y 370.916,Z 298.616,A -85,B 0,C 180,E1 -12711.481,E2 -12711.481} C_VEL
LIN {X 0,Y 371.684,Z 289.72,A -85,B 0,C 180,E1 -12713.691,E2 -12713.691} C_VEL
LIN {X 0,Y 370.687,Z 282.783,A -85,B 0,C 180,E1 -12715.551,E2 -12715.551} C_VEL
LIN {X 0,Y 368.976,Z 274.335,A -85,B 0,C 180,E1 -12717.972,E2 -12717.972} C_VEL
LIN {X 0,Y 368.919,Z 274.345,A -85,B 0,C 180,E1 -12720.986,E2 -12720.986} C_VEL
LIN {X 0,Y 368.939,Z 274.34,A -85,B 0,C 180,E1 -12724.853,E2 -12724.853} C_VEL
LIN {X 0,Y 368.887,Z 274.346,A -85,B 0,C 180,E1 -12728.633,E2 -12728.633} C_VEL
LIN {X 0,Y 368.886,Z 274.347,A -85,B 0,C 180,E1 -12732.007,E2 -12732.007} C_VEL
LIN {X 0,Y 368.887,Z 274.345,A -85,B 0,C 180,E1 -12735.174,E2 -12735.174} C_VEL
LIN {X 0,Y 368.879,Z 274.346,A -85,B 0,C 180,E1 -12738.174,E2 -12738.174} C_VEL
LIN {X 0,Y 368.885,Z 274.343,A -85,B 0,C 180,E1 -12741.364,E2 -12741.364} C_VEL
LIN {X 0,Y 368.944,Z 274.333,A -85,B 0,C 180,E1 -12745.144,E2 -12745.144} C_VEL
LIN {X 0,Y 368.92,Z 274.336,A -85,B 0,C 180,E1 -12749.043,E2 -12749.043} C_VEL
LIN {X 0,Y 368.923,Z 274.345,A -85,B 0,C 180,E1 -12751.556,E2 -12751.556} C_VEL
LIN {X 0,Y 368.941,Z 274.337,A -85,B 0,C 180,E1 -12755.221,E2 -12755.221} C_VEL
LIN {X 0,Y 368.926,Z 274.332,A -85,B 0,C 180,E1 -12758.978,E2 -12758.978} C_VEL
LIN {X 0,Y 368.996,Z 274.328,A -85,B 0,C 180,E1 -12762.254,E2 -12762.254} C_VEL
LIN {X 0,Y 369.042,Z 274.326,A -85,B 0,C 180,E1 -12766.225,E2 -12766.225} C_VEL
LIN {X 0,Y 369.07,Z 274.318,A -85,B 0,C 180,E1 -12770.129,E2 -12770.129} C_VEL
LIN {X 0,Y 369.201,Z 274.301,A -85,B 0,C 180,E1 -12773.438,E2 -12773.438} C_VEL
LIN {X 0,Y 369.309,Z 274.292,A -85,B 0,C 180,E1 -12777.815,E2 -12777.815} C_VEL
LIN {X 0,Y 369.453,Z 274.267,A -85,B 0,C 180,E1 -12779.996,E2 -12779.996} C_VEL
LIN {X 0,Y 369.313,Z 274.293,A -85,B 0,C 180,E1 -12782.178,E2 -12782.178} C_VEL
LIN {X 0,Y 369.17,Z 274.31,A -85,B 0,C 180,E1 -12786.555,E2 -12786.555} C_VEL
LIN {X 0,Y 369.059,Z 274.322,A -85,B 0,C 180,E1 -12789.865,E2 -12789.865} C_VEL
LIN {X 0,Y 369.031,Z 274.328,A -85,B 0,C 180,E1 -12793.768,E2 -12793.768} C_VEL
LIN {X 0,Y 368.993,Z 274.332,A -85,B 0,C 180,E1 -12797.764,E2 -12797.764} C_VEL
LIN {X 0,Y 368.919,Z 274.338,A -85,B 0,C 180,E1 -12801.216,E2 -12801.216} C_VEL
LIN {X 0,Y 368.946,Z 274.336,A -85,B 0,C 180,E1 -12804.771,E2 -12804.771} C_VEL
LIN {X 0,Y 368.95,Z 274.337,A -85,B 0,C 180,E1 -12807.199,E2 -12807.199} C_VEL
LIN {X 0,Y 368.914,Z 274.341,A -85,B 0,C 180,E1 -12810.95,E2 -12810.95} C_VEL
LIN {X 0,Y 368.911,Z 274.334,A -85,B 0,C 180,E1 -12814.998,E2 -12814.998} C_VEL
LIN {X 0,Y 368.889,Z 274.349,A -85,B 0,C 180,E1 -12818.637,E2 -12818.637} C_VEL
LIN {X 0,Y 368.919,Z 274.343,A -85,B 0,C 180,E1 -12822.016,E2 -12822.016} C_VEL
LIN {X 0,Y 368.967,Z 274.339,A -85,B 0,C 180,E1 -12825.189,E2 -12825.189} C_VEL
LIN {X 0,Y 368.916,Z 274.344,A -85,B 0,C 180,E1 -12828.182,E2 -12828.182} C_VEL
LIN {X 0,Y 368.887,Z 274.349,A -85,B 0,C 180,E1 -12831.356,E2 -12831.356} C_VEL
LIN {X 0,Y 368.894,Z 274.41,A -85,B 0,C 180,E1 -12832.898,E2 -12832.898} C_VEL
LIN {X 0,Y 370.451,Z 282.206,A -85,B 0,C 180,E1 -12835.238,E2 -12835.238} C_VEL
LIN {X 0,Y 374.281,Z 297.889,A -85,B 0,C 180,E1 -12835.814,E2 -12835.814} C_VEL
LIN {X 0,Y 375.077,Z 303.405,A -85,B 0,C 180,E1 -12835.973,E2 -12835.973} C_VEL
LIN {X 0,Y 374.133,Z 359.271,A -85,B 0,C 180,E1 -12837.092,E2 -12837.092} C_VEL
LIN {X 0,Y 373.816,Z 369.476,A -85,B 0,C 180,E1 -12837.459,E2 -12837.459} C_VEL
LIN {X 0,Y 373.322,Z 380.818,A -85,B 0,C 180,E1 -12838.081,E2 -12838.081} C_VEL
LIN {X 0,Y 372.72,Z 389.839,A -85,B 0,C 180,E1 -12838.766,E2 -12838.766} C_VEL
LIN {X 0,Y 372.007,Z 398.863,A -85,B 0,C 180,E1 -12839.645,E2 -12839.645} C_VEL
LIN {X 0,Y 371.342,Z 406.172,A -85,B 0,C 180,E1 -12840.523,E2 -12840.523} C_VEL
LIN {X 0,Y 370.722,Z 412.284,A -85,B 0,C 180,E1 -12841.401,E2 -12841.401} C_VEL
LIN {X 0,Y 369.991,Z 419.008,A -85,B 0,C 180,E1 -12842.572,E2 -12842.572} C_VEL
LIN {X 0,Y 369.433,Z 424.239,A -85,B 0,C 180,E1 -12843.681,E2 -12843.681} C_VEL
LIN {X 0,Y 368.923,Z 429.038,A -85,B 0,C 180,E1 -12844.921,E2 -12844.921} C_VEL
LIN {X 0,Y 368.4,Z 433.51,A -85,B 0,C 180,E1 -12846.383,E2 -12846.383} C_VEL
LIN {X 0,Y 368.079,Z 436.257,A -85,B 0,C 180,E1 -12847.55,E2 -12847.55} C_VEL
LIN {X 0,Y 367.838,Z 438.364,A -85,B 0,C 180,E1 -12848.715,E2 -12848.715} C_VEL
LIN {X 0,Y 367.622,Z 439.888,A -85,B 0,C 180,E1 -12849.872,E2 -12849.872} C_VEL
LIN {X 0,Y 367.463,Z 440.846,A -85,B 0,C 180,E1 -12851.026,E2 -12851.026} C_VEL
LIN {X 0,Y 367.399,Z 441.181,A -85,B 0,C 180,E1 -12852.178,E2 -12852.178} C_VEL
LIN {X 0,Y 367.411,Z 440.969,A -85,B 0,C 180,E1 -12853.326,E2 -12853.326} C_VEL
LIN {X 0,Y 367.41,Z 440.251,A -85,B 0,C 180,E1 -12854.467,E2 -12854.467} C_VEL
LIN {X 0,Y 367.498,Z 439.014,A -85,B 0,C 180,E1 -12855.605,E2 -12855.605} C_VEL
LIN {X 0,Y 367.689,Z 436.506,A -85,B 0,C 180,E1 -12857.088,E2 -12857.088} C_VEL
LIN {X 0,Y 367.866,Z 433.357,A -85,B 0,C 180,E1 -12858.428,E2 -12858.428} C_VEL
LIN {X 0,Y 368.231,Z 428.059,A -85,B 0,C 180,E1 -12860.109,E2 -12860.109} C_VEL
LIN {X 0,Y 368.647,Z 421.048,A -85,B 0,C 180,E1 -12861.78,E2 -12861.78} C_VEL
LIN {X 0,Y 369.111,Z 415.095,A -85,B 0,C 180,E1 -12862.891,E2 -12862.891} C_VEL
LIN {X 0,Y 369.571,Z 407.861,A -85,B 0,C 180,E1 -12863.997,E2 -12863.997} C_VEL
LIN {X 0,Y 370.107,Z 400.124,A -85,B 0,C 180,E1 -12864.962,E2 -12864.962} C_VEL
LIN {X 0,Y 370.58,Z 392.009,A -85,B 0,C 180,E1 -12865.786,E2 -12865.786} C_VEL
LIN {X 0,Y 370.979,Z 383.604,A -85,B 0,C 180,E1 -12866.47,E2 -12866.47} C_VEL
LIN {X 0,Y 371.313,Z 375.02,A -85,B 0,C 180,E1 -12867.017,E2 -12867.017} C_VEL
LIN {X 0,Y 371.631,Z 364.772,A -85,B 0,C 180,E1 -12867.494,E2 -12867.494} C_VEL
LIN {X 0,Y 371.858,Z 351.029,A -85,B 0,C 180,E1 -12867.868,E2 -12867.868} C_VEL
LIN {X 0,Y 372.417,Z 299.976,A -85,B 0,C 180,E1 -12868.851,E2 -12868.851} C_VEL
LIN {X 0,Y 369.384,Z 281.968,A -85,B 0,C 180,E1 -12869.319,E2 -12869.319} C_VEL
LIN {X 0,Y 369.441,Z 275.663,A -85,B 0,C 180,E1 -12871.09,E2 -12871.09} C_VEL
LIN {X 0,Y 369.27,Z 274.299,A -85,B 0,C 180,E1 -12871.5,E2 -12871.5} C_VEL
LIN {X 0,Y 369.165,Z 274.31,A -85,B 0,C 180,E1 -12876.559,E2 -12876.559} C_VEL
LIN {X 0,Y 369.032,Z 274.326,A -85,B 0,C 180,E1 -12879.869,E2 -12879.869} C_VEL
LIN {X 0,Y 368.997,Z 274.331,A -85,B 0,C 180,E1 -12883.858,E2 -12883.858} C_VEL
LIN {X 0,Y 368.299,Z 274.42,A -85,B 0,C 180,E1 -12884.769,E2 -12884.769} C_VEL
LIN {X 0,Y 365.435,Z 274.773,A -85,B 0,C 180,E1 -12886.251,E2 -12886.251} C_VEL
LIN {X 0,Y 363.02,Z 275.08,A -85,B 0,C 180,E1 -12887.449,E2 -12887.449} C_VEL
LIN {X 0,Y 361.972,Z 275.205,A -85,B 0,C 180,E1 -12888.376,E2 -12888.376} C_VEL
LIN {X 0,Y 361.879,Z 275.217,A -85,B 0,C 180,E1 -12888.69,E2 -12888.69} C_VEL
LIN {X 0,Y 361.858,Z 275.223,A -85,B 0,C 180,E1 -12891.655,E2 -12891.655} C_VEL
LIN {X 0,Y 361.852,Z 275.225,A -85,B 0,C 180,E1 -12895.296,E2 -12895.296} C_VEL
LIN {X 0,Y 361.826,Z 275.225,A -85,B 0,C 180,E1 -12899.076,E2 -12899.076} C_VEL
LIN {X 0,Y 361.82,Z 275.225,A -85,B 0,C 180,E1 -12902.948,E2 -12902.948} C_VEL
LIN {X 0,Y 361.841,Z 275.227,A -85,B 0,C 180,E1 -12905.64,E2 -12905.64} C_VEL
LIN {X 0,Y 361.8,Z 275.227,A -85,B 0,C 180,E1 -12909.021,E2 -12909.021} C_VEL
LIN {X 0,Y 361.81,Z 275.225,A -85,B 0,C 180,E1 -12912.833,E2 -12912.833} C_VEL
LIN {X 0,Y 361.797,Z 275.231,A -85,B 0,C 180,E1 -12915.951,E2 -12915.951} C_VEL
LIN {X 0,Y 361.815,Z 275.226,A -85,B 0,C 180,E1 -12919.249,E2 -12919.249} C_VEL
LIN {X 0,Y 361.845,Z 275.221,A -85,B 0,C 180,E1 -12922.782,E2 -12922.782} C_VEL
LIN {X 0,Y 361.839,Z 275.227,A -85,B 0,C 180,E1 -12925.724,E2 -12925.724} C_VEL
LIN {X 0,Y 361.843,Z 275.225,A -85,B 0,C 180,E1 -12929.675,E2 -12929.675} C_VEL
LIN {X 0,Y 361.856,Z 275.221,A -85,B 0,C 180,E1 -12933.472,E2 -12933.472} C_VEL
LIN {X 0,Y 361.869,Z 275.218,A -85,B 0,C 180,E1 -12937.148,E2 -12937.148} C_VEL
LIN {X 0,Y 361.919,Z 275.213,A -85,B 0,C 180,E1 -12940.729,E2 -12940.729} C_VEL
LIN {X 0,Y 362.06,Z 275.34,A -85,B 0,C 180,E1 -12942.613,E2 -12942.613} C_VEL
LIN {X 0,Y 361.989,Z 281.107,A -85,B 0,C 180,E1 -12944.124,E2 -12944.124} C_VEL
LIN {X 0,Y 364.6,Z 301.097,A -85,B 0,C 180,E1 -12944.731,E2 -12944.731} C_VEL
LIN {X 0,Y 363.445,Z 360.192,A -85,B 0,C 180,E1 -12946.302,E2 -12946.302} C_VEL
LIN {X 0,Y 363.261,Z 369.936,A -85,B 0,C 180,E1 -12946.722,E2 -12946.722} C_VEL
LIN {X 0,Y 362.915,Z 380.468,A -85,B 0,C 180,E1 -12947.35,E2 -12947.35} C_VEL
LIN {X 0,Y 362.538,Z 391.704,A -85,B 0,C 180,E1 -12948.26,E2 -12948.26} C_VEL
LIN {X 0,Y 362.103,Z 400.996,A -85,B 0,C 180,E1 -12949.237,E2 -12949.237} C_VEL
LIN {X 0,Y 361.654,Z 409.598,A -85,B 0,C 180,E1 -12950.355,E2 -12950.355} C_VEL
LIN {X 0,Y 361.264,Z 417.395,A -85,B 0,C 180,E1 -12951.614,E2 -12951.614} C_VEL
LIN {X 0,Y 360.998,Z 424.232,A -85,B 0,C 180,E1 -12953.015,E2 -12953.015} C_VEL
LIN {X 0,Y 360.771,Z 428.525,A -85,B 0,C 180,E1 -12954.079,E2 -12954.079} C_VEL
LIN {X 0,Y 360.669,Z 433.223,A -85,B 0,C 180,E1 -12955.533,E2 -12955.533} C_VEL
LIN {X 0,Y 360.524,Z 436.064,A -85,B 0,C 180,E1 -12956.651,E2 -12956.651} C_VEL
LIN {X 0,Y 360.439,Z 438.294,A -85,B 0,C 180,E1 -12957.769,E2 -12957.769} C_VEL
LIN {X 0,Y 360.436,Z 439.956,A -85,B 0,C 180,E1 -12958.886,E2 -12958.886} C_VEL
LIN {X 0,Y 360.464,Z 441.032,A -85,B 0,C 180,E1 -12960.004,E2 -12960.004} C_VEL
LIN {X 0,Y 360.511,Z 441.507,A -85,B 0,C 180,E1 -12961.121,E2 -12961.121} C_VEL
LIN {X 0,Y 360.639,Z 441.44,A -85,B 0,C 180,E1 -12962.237,E2 -12962.237} C_VEL
LIN {X 0,Y 360.877,Z 440.846,A -85,B 0,C 180,E1 -12963.353,E2 -12963.353} C_VEL
LIN {X 0,Y 361.158,Z 439.73,A -85,B 0,C 180,E1 -12964.468,E2 -12964.468} C_VEL
LIN {X 0,Y 361.375,Z 438.086,A -85,B 0,C 180,E1 -12965.584,E2 -12965.584} C_VEL
LIN {X 0,Y 361.416,Z 435.855,A -85,B 0,C 180,E1 -12966.704,E2 -12966.704} C_VEL
LIN {X 0,Y 362.237,Z 431.353,A -85,B 0,C 180,E1 -12968.314,E2 -12968.314} C_VEL
LIN {X 0,Y 362.856,Z 426.079,A -85,B 0,C 180,E1 -12969.761,E2 -12969.761} C_VEL
LIN {X 0,Y 363.681,Z 419.679,A -85,B 0,C 180,E1 -12971.145,E2 -12971.145} C_VEL
LIN {X 0,Y 364.685,Z 411.594,A -85,B 0,C 180,E1 -12972.525,E2 -12972.525} C_VEL
LIN {X 0,Y 365.582,Z 403.49,A -85,B 0,C 180,E1 -12973.624,E2 -12973.624} C_VEL
LIN {X 0,Y 366.418,Z 394.806,A -85,B 0,C 180,E1 -12974.584,E2 -12974.584} C_VEL
LIN {X 0,Y 367.363,Z 383.771,A -85,B 0,C 180,E1 -12975.538,E2 -12975.538} C_VEL
LIN {X 0,Y 368.042,Z 372.988,A -85,B 0,C 180,E1 -12976.22,E2 -12976.22} C_VEL
LIN {X 0,Y 368.635,Z 361.434,A -85,B 0,C 180,E1 -12976.742,E2 -12976.742} C_VEL
LIN {X 0,Y 371,Z 304.7,A -85,B 0,C 180,E1 -12978.429,E2 -12978.429} C_VEL
LIN {X 0,Y 367.818,Z 292.531,A -85,B 0,C 180,E1 -12979.157,E2 -12979.157} C_VEL
LIN {X 0,Y 364.201,Z 284.332,A -85,B 0,C 180,E1 -12979.847,E2 -12979.847} C_VEL
LIN {X 0,Y 361.888,Z 275.223,A -85,B 0,C 180,E1 -12982.708,E2 -12982.708} C_VEL
LIN {X 0,Y 361.875,Z 275.221,A -85,B 0,C 180,E1 -12986.534,E2 -12986.534} C_VEL
LIN {X 0,Y 361.866,Z 275.224,A -85,B 0,C 180,E1 -12990.332,E2 -12990.332} C_VEL
LIN {X 0,Y 361.86,Z 275.224,A -85,B 0,C 180,E1 -12994.283,E2 -12994.283} C_VEL
LIN {X 0,Y 361.868,Z 275.222,A -85,B 0,C 180,E1 -12997.223,E2 -12997.223} C_VEL
LIN {X 0,Y 361.822,Z 275.228,A -85,B 0,C 180,E1 -13000.752,E2 -13000.752} C_VEL
LIN {X 0,Y 361.827,Z 275.226,A -85,B 0,C 180,E1 -13004.37,E2 -13004.37} C_VEL
LIN {X 0,Y 361.844,Z 275.221,A -85,B 0,C 180,E1 -13007.57,E2 -13007.57} C_VEL
LIN {X 0,Y 361.839,Z 275.226,A -85,B 0,C 180,E1 -13010.982,E2 -13010.982} C_VEL
LIN {X 0,Y 361.883,Z 275.221,A -85,B 0,C 180,E1 -13014.657,E2 -13014.657} C_VEL
LIN {X 0,Y 361.847,Z 275.221,A -85,B 0,C 180,E1 -13018.371,E2 -13018.371} C_VEL
LIN {X 0,Y 361.921,Z 275.216,A -85,B 0,C 180,E1 -13022.222,E2 -13022.222} C_VEL
LIN {X 0,Y 361.989,Z 275.331,A -85,B 0,C 180,E1 -13023.71,E2 -13023.71} C_VEL
LIN {X 0,Y 363.666,Z 285.395,A -85,B 0,C 180,E1 -13026.359,E2 -13026.359} C_VEL
LIN {X 0,Y 363.172,Z 293.705,A -85,B 0,C 180,E1 -13028.427,E2 -13028.427} C_VEL
LIN {X 0,Y 362.737,Z 299.763,A -85,B 0,C 180,E1 -13029.914,E2 -13029.914} C_VEL
LIN {X 0,Y 363.27,Z 303.428,A -85,B 0,C 180,E1 -13030.173,E2 -13030.173} C_VEL
LIN {X 0,Y 366.564,Z 321.004,A -85,B 0,C 180,E1 -13031.135,E2 -13031.135} C_VEL
LIN {X 0,Y 368.648,Z 336.022,A -85,B 0,C 180,E1 -13031.84,E2 -13031.84} C_VEL
LIN {X 0,Y 369.262,Z 348.028,A -85,B 0,C 180,E1 -13032.303,E2 -13032.303} C_VEL
LIN {X 0,Y 367.399,Z 393.737,A -85,B 0,C 180,E1 -13033.682,E2 -13033.682} C_VEL
LIN {X 0,Y 366.45,Z 406.18,A -85,B 0,C 180,E1 -13034.282,E2 -13034.282} C_VEL
LIN {X 0,Y 365.587,Z 416.112,A -85,B 0,C 180,E1 -13034.958,E2 -13034.958} C_VEL
LIN {X 0,Y 364.682,Z 425.471,A -85,B 0,C 180,E1 -13035.776,E2 -13035.776} C_VEL
LIN {X 0,Y 363.615,Z 435.264,A -85,B 0,C 180,E1 -13036.873,E2 -13036.873} C_VEL
LIN {X 0,Y 362.78,Z 443.095,A -85,B 0,C 180,E1 -13037.98,E2 -13037.98} C_VEL
LIN {X 0,Y 362.07,Z 449.617,A -85,B 0,C 180,E1 -13039.091,E2 -13039.091} C_VEL
LIN {X 0,Y 361.515,Z 455.048,A -85,B 0,C 180,E1 -13040.206,E2 -13040.206} C_VEL
LIN {X 0,Y 360.992,Z 460.589,A -85,B 0,C 180,E1 -13041.604,E2 -13041.604} C_VEL
LIN {X 0,Y 360.59,Z 465.726,A -85,B 0,C 180,E1 -13043.284,E2 -13043.284} C_VEL
LIN {X 0,Y 360.434,Z 468.268,A -85,B 0,C 180,E1 -13044.405,E2 -13044.405} C_VEL
LIN {X 0,Y 360.431,Z 470.187,A -85,B 0,C 180,E1 -13045.526,E2 -13045.526} C_VEL
LIN {X 0,Y 360.404,Z 473.005,A -85,B 0,C 180,E1 -13047.765,E2 -13047.765} C_VEL
LIN {X 0,Y 360.48,Z 474.009,A -85,B 0,C 180,E1 -13048.883,E2 -13048.883} C_VEL
LIN {X 0,Y 360.482,Z 474.52,A -85,B 0,C 180,E1 -13050,E2 -13050} C_VEL
LIN {X 0,Y 360.437,Z 474.563,A -85,B 0,C 180,E1 -13051.117,E2 -13051.117} C_VEL
LIN {X 0,Y 360.357,Z 474.141,A -85,B 0,C 180,E1 -13052.235,E2 -13052.235} C_VEL
LIN {X 0,Y 360.347,Z 473.149,A -85,B 0,C 180,E1 -13053.354,E2 -13053.354} C_VEL
LIN {X 0,Y 360.423,Z 470.728,A -85,B 0,C 180,E1 -13055.034,E2 -13055.034} C_VEL
LIN {X 0,Y 360.596,Z 466.982,A -85,B 0,C 180,E1 -13056.715,E2 -13056.715} C_VEL
LIN {X 0,Y 360.872,Z 463.798,A -85,B 0,C 180,E1 -13057.835,E2 -13057.835} C_VEL
LIN {X 0,Y 361.295,Z 458.754,A -85,B 0,C 180,E1 -13059.235,E2 -13059.235} C_VEL
LIN {X 0,Y 361.954,Z 452.437,A -85,B 0,C 180,E1 -13060.629,E2 -13060.629} C_VEL
LIN {X 0,Y 362.615,Z 446.27,A -85,B 0,C 180,E1 -13061.742,E2 -13061.742} C_VEL
LIN {X 0,Y 363.287,Z 439.807,A -85,B 0,C 180,E1 -13062.712,E2 -13062.712} C_VEL
LIN {X 0,Y 363.976,Z 433.228,A -85,B 0,C 180,E1 -13063.54,E2 -13063.54} C_VEL
LIN {X 0,Y 364.714,Z 425.281,A -85,B 0,C 180,E1 -13064.365,E2 -13064.365} C_VEL
LIN {X 0,Y 365.486,Z 417.091,A -85,B 0,C 180,E1 -13065.046,E2 -13065.046} C_VEL
LIN {X 0,Y 366.063,Z 408.825,A -85,B 0,C 180,E1 -13065.592,E2 -13065.592} C_VEL
LIN {X 0,Y 366.616,Z 400.309,A -85,B 0,C 180,E1 -13066.015,E2 -13066.015} C_VEL
LIN {X 0,Y 367.074,Z 390.546,A -85,B 0,C 180,E1 -13066.346,E2 -13066.346} C_VEL
LIN {X 0,Y 367.708,Z 343.937,A -85,B 0,C 180,E1 -13067.304,E2 -13067.304} C_VEL
LIN {X 0,Y 365.289,Z 326.619,A -85,B 0,C 180,E1 -13067.811,E2 -13067.811} C_VEL
LIN {X 0,Y 362.824,Z 313.174,A -85,B 0,C 180,E1 -13068.26,E2 -13068.26} C_VEL
LIN {X 0,Y 364.081,Z 298.461,A -85,B 0,C 180,E1 -13071.939,E2 -13071.939} C_VEL
LIN {X 0,Y 364.749,Z 290.854,A -85,B 0,C 180,E1 -13073.868,E2 -13073.868} C_VEL
LIN {X 0,Y 363.715,Z 283.919,A -85,B 0,C 180,E1 -13075.77,E2 -13075.77} C_VEL
LIN {X 0,Y 361.949,Z 275.212,A -85,B 0,C 180,E1 -13078.327,E2 -13078.327} C_VEL
LIN {X 0,Y 361.846,Z 275.221,A -85,B 0,C 180,E1 -13081.628,E2 -13081.628} C_VEL
LIN {X 0,Y 361.878,Z 275.214,A -85,B 0,C 180,E1 -13085.342,E2 -13085.342} C_VEL
LIN {X 0,Y 361.838,Z 275.224,A -85,B 0,C 180,E1 -13089.017,E2 -13089.017} C_VEL
LIN {X 0,Y 361.844,Z 275.224,A -85,B 0,C 180,E1 -13092.827,E2 -13092.827} C_VEL
LIN {X 0,Y 361.826,Z 275.227,A -85,B 0,C 180,E1 -13095.945,E2 -13095.945} C_VEL
LIN {X 0,Y 361.821,Z 275.228,A -85,B 0,C 180,E1 -13099.247,E2 -13099.247} C_VEL
LIN {X 0,Y 361.872,Z 275.219,A -85,B 0,C 180,E1 -13102.98,E2 -13102.98} C_VEL
LIN {X 0,Y 361.866,Z 275.219,A -85,B 0,C 180,E1 -13106.629,E2 -13106.629} C_VEL
LIN {X 0,Y 361.864,Z 275.217,A -85,B 0,C 180,E1 -13109.668,E2 -13109.668} C_VEL
LIN {X 0,Y 361.886,Z 275.214,A -85,B 0,C 180,E1 -13113.467,E2 -13113.467} C_VEL
LIN {X 0,Y 361.885,Z 275.217,A -85,B 0,C 180,E1 -13117.141,E2 -13117.141} C_VEL
LIN {X 0,Y 361.892,Z 275.215,A -85,B 0,C 180,E1 -13120.72,E2 -13120.72} C_VEL
LIN {X 0,Y 361.948,Z 275.204,A -85,B 0,C 180,E1 -13124.223,E2 -13124.223} C_VEL
LIN {X 0,Y 362.003,Z 275.2,A -85,B 0,C 180,E1 -13126.525,E2 -13126.525} C_VEL
LIN {X 0,Y 362.034,Z 275.191,A -85,B 0,C 180,E1 -13129.935,E2 -13129.935} C_VEL
LIN {X 0,Y 362.163,Z 275.177,A -85,B 0,C 180,E1 -13133.31,E2 -13133.31} C_VEL
LIN {X 0,Y 362.272,Z 275.168,A -85,B 0,C 180,E1 -13137.773,E2 -13137.773} C_VEL
LIN {X 0,Y 362.402,Z 275.144,A -85,B 0,C 180,E1 -13139.996,E2 -13139.996} C_VEL
LIN {X 0,Y 362.277,Z 275.17,A -85,B 0,C 180,E1 -13142.22,E2 -13142.22} C_VEL
LIN {X 0,Y 362.132,Z 275.186,A -85,B 0,C 180,E1 -13146.683,E2 -13146.683} C_VEL
LIN {X 0,Y 361.996,Z 275.2,A -85,B 0,C 180,E1 -13150.059,E2 -13150.059} C_VEL
LIN {X 0,Y 361.992,Z 275.206,A -85,B 0,C 180,E1 -13153.895,E2 -13153.895} C_VEL
LIN {X 0,Y 361.959,Z 275.209,A -85,B 0,C 180,E1 -13157.935,E2 -13157.935} C_VEL
LIN {X 0,Y 361.882,Z 275.215,A -85,B 0,C 180,E1 -13161.649,E2 -13161.649} C_VEL
LIN {X 0,Y 361.916,Z 275.211,A -85,B 0,C 180,E1 -13165.286,E2 -13165.286} C_VEL
LIN {X 0,Y 361.895,Z 275.216,A -85,B 0,C 180,E1 -13167.775,E2 -13167.775} C_VEL
LIN {X 0,Y 361.821,Z 275.222,A -85,B 0,C 180,E1 -13171.625,E2 -13171.625} C_VEL
LIN {X 0,Y 361.856,Z 275.211,A -85,B 0,C 180,E1 -13175.341,E2 -13175.341} C_VEL
LIN {X 0,Y 361.851,Z 275.221,A -85,B 0,C 180,E1 -13179.023,E2 -13179.023} C_VEL
LIN {X 0,Y 361.864,Z 275.225,A -85,B 0,C 180,E1 -13182.437,E2 -13182.437} C_VEL
LIN {X 0,Y 361.906,Z 275.217,A -85,B 0,C 180,E1 -13185.925,E2 -13185.925} C_VEL
LIN {X 0,Y 361.88,Z 275.219,A -85,B 0,C 180,E1 -13189.229,E2 -13189.229} C_VEL
LIN {X 0,Y 361.879,Z 275.381,A -85,B 0,C 180,E1 -13192.596,E2 -13192.596} C_VEL
LIN {X 0,Y 363.345,Z 282.654,A -85,B 0,C 180,E1 -13194.816,E2 -13194.816} C_VEL
LIN {X 0,Y 366.123,Z 292.211,A -85,B 0,C 180,E1 -13195.197,E2 -13195.197} C_VEL
LIN {X 0,Y 368.466,Z 303.136,A -85,B 0,C 180,E1 -13195.573,E2 -13195.573} C_VEL
LIN {X 0,Y 367.466,Z 358.897,A -85,B 0,C 180,E1 -13196.705,E2 -13196.705} C_VEL
LIN {X 0,Y 367.228,Z 368.101,A -85,B 0,C 180,E1 -13197.028,E2 -13197.028} C_VEL
LIN {X 0,Y 366.764,Z 378.242,A -85,B 0,C 180,E1 -13197.552,E2 -13197.552} C_VEL
LIN {X 0,Y 366.062,Z 388.693,A -85,B 0,C 180,E1 -13198.294,E2 -13198.294} C_VEL
LIN {X 0,Y 365.324,Z 398.023,A -85,B 0,C 180,E1 -13199.189,E2 -13199.189} C_VEL
LIN {X 0,Y 364.585,Z 406.036,A -85,B 0,C 180,E1 -13200.153,E2 -13200.153} C_VEL
LIN {X 0,Y 363.842,Z 412.714,A -85,B 0,C 180,E1 -13201.125,E2 -13201.125} C_VEL
LIN {X 0,Y 363.09,Z 419.424,A -85,B 0,C 180,E1 -13202.319,E2 -13202.319} C_VEL
LIN {X 0,Y 362.456,Z 424.919,A -85,B 0,C 180,E1 -13203.515,E2 -13203.515} C_VEL
LIN {X 0,Y 361.941,Z 429.425,A -85,B 0,C 180,E1 -13204.711,E2 -13204.711} C_VEL
LIN {X 0,Y 361.448,Z 433.432,A -85,B 0,C 180,E1 -13206.032,E2 -13206.032} C_VEL
LIN {X 0,Y 360.979,Z 437.223,A -85,B 0,C 180,E1 -13207.688,E2 -13207.688} C_VEL
LIN {X 0,Y 360.624,Z 439.955,A -85,B 0,C 180,E1 -13209.464,E2 -13209.464} C_VEL
LIN {X 0,Y 360.416,Z 440.973,A -85,B 0,C 180,E1 -13210.641,E2 -13210.641} C_VEL
LIN {X 0,Y 360.314,Z 441.437,A -85,B 0,C 180,E1 -13211.815,E2 -13211.815} C_VEL
LIN {X 0,Y 360.293,Z 441.383,A -85,B 0,C 180,E1 -13212.987,E2 -13212.987} C_VEL
LIN {X 0,Y 360.309,Z 440.818,A -85,B 0,C 180,E1 -13214.153,E2 -13214.153} C_VEL
LIN {X 0,Y 360.372,Z 439.737,A -85,B 0,C 180,E1 -13215.314,E2 -13215.314} C_VEL
LIN {X 0,Y 360.584,Z 437.007,A -85,B 0,C 180,E1 -13217.015,E2 -13217.015} C_VEL
LIN {X 0,Y 360.85,Z 432.855,A -85,B 0,C 180,E1 -13218.769,E2 -13218.769} C_VEL
LIN {X 0,Y 361.094,Z 429.301,A -85,B 0,C 180,E1 -13219.912,E2 -13219.912} C_VEL
LIN {X 0,Y 361.388,Z 425.004,A -85,B 0,C 180,E1 -13221.05,E2 -13221.05} C_VEL
LIN {X 0,Y 361.753,Z 419.829,A -85,B 0,C 180,E1 -13222.184,E2 -13222.184} C_VEL
LIN {X 0,Y 362.171,Z 413.589,A -85,B 0,C 180,E1 -13223.314,E2 -13223.314} C_VEL
LIN {X 0,Y 362.623,Z 407.022,A -85,B 0,C 180,E1 -13224.3,E2 -13224.3} C_VEL
LIN {X 0,Y 363.175,Z 399.054,A -85,B 0,C 180,E1 -13225.283,E2 -13225.283} C_VEL
LIN {X 0,Y 363.669,Z 390.635,A -85,B 0,C 180,E1 -13226.122,E2 -13226.122} C_VEL
LIN {X 0,Y 364.226,Z 379.819,A -85,B 0,C 180,E1 -13226.958,E2 -13226.958} C_VEL
LIN {X 0,Y 364.598,Z 368.817,A -85,B 0,C 180,E1 -13227.549,E2 -13227.549} C_VEL
LIN {X 0,Y 364.795,Z 358.896,A -85,B 0,C 180,E1 -13227.906,E2 -13227.906} C_VEL
LIN {X 0,Y 365.466,Z 300.524,A -85,B 0,C 180,E1 -13229.087,E2 -13229.087} C_VEL
LIN {X 0,Y 362.403,Z 282.221,A -85,B 0,C 180,E1 -13229.583,E2 -13229.583} C_VEL
LIN {X 0,Y 362.447,Z 276.869,A -85,B 0,C 180,E1 -13231.111,E2 -13231.111} C_VEL
LIN {X 0,Y 362.252,Z 275.172,A -85,B 0,C 180,E1 -13231.668,E2 -13231.668} C_VEL
LIN {X 0,Y 362.127,Z 275.187,A -85,B 0,C 180,E1 -13236.687,E2 -13236.687} C_VEL
LIN {X 0,Y 361.996,Z 275.202,A -85,B 0,C 180,E1 -13240.063,E2 -13240.063} C_VEL
LIN {X 0,Y 361.964,Z 275.207,A -85,B 0,C 180,E1 -13243.9,E2 -13243.9} C_VEL
LIN {X 0,Y 361.935,Z 275.211,A -85,B 0,C 180,E1 -13247.94,E2 -13247.94} C_VEL
LIN {X 0,Y 361.879,Z 275.217,A -85,B 0,C 180,E1 -13248.69,E2 -13248.69} C_VEL
LIN {X 0,Y 361.189,Z 275.309,A -85,B 0,C 180,E1 -13249.619,E2 -13249.619} C_VEL
LIN {X 0,Y 358.318,Z 275.671,A -85,B 0,C 180,E1 -13251.129,E2 -13251.129} C_VEL
LIN {X 0,Y 355.9,Z 275.972,A -85,B 0,C 180,E1 -13252.351,E2 -13252.351} C_VEL
LIN {X 0,Y 354.865,Z 276.096,A -85,B 0,C 180,E1 -13253.297,E2 -13253.297} C_VEL
LIN {X 0,Y 354.781,Z 276.103,A -85,B 0,C 180,E1 -13253.617,E2 -13253.617} C_VEL
LIN {X 0,Y 354.776,Z 276.104,A -85,B 0,C 180,E1 -13257.105,E2 -13257.105} C_VEL
LIN {X 0,Y 354.767,Z 276.107,A -85,B 0,C 180,E1 -13259.687,E2 -13259.687} C_VEL
LIN {X 0,Y 354.759,Z 276.104,A -85,B 0,C 180,E1 -13262.337,E2 -13262.337} C_VEL
LIN {X 0,Y 354.795,Z 276.104,A -85,B 0,C 180,E1 -13265.702,E2 -13265.702} C_VEL
LIN {X 0,Y 354.743,Z 276.109,A -85,B 0,C 180,E1 -13269.416,E2 -13269.416} C_VEL
LIN {X 0,Y 354.762,Z 276.103,A -85,B 0,C 180,E1 -13272.87,E2 -13272.87} C_VEL
LIN {X 0,Y 354.746,Z 276.108,A -85,B 0,C 180,E1 -13276.107,E2 -13276.107} C_VEL
LIN {X 0,Y 354.768,Z 276.104,A -85,B 0,C 180,E1 -13279.183,E2 -13279.183} C_VEL
LIN {X 0,Y 354.789,Z 276.101,A -85,B 0,C 180,E1 -13282.407,E2 -13282.407} C_VEL
LIN {X 0,Y 354.796,Z 276.099,A -85,B 0,C 180,E1 -13284.945,E2 -13284.945} C_VEL
LIN {X 0,Y 354.779,Z 276.103,A -85,B 0,C 180,E1 -13288.409,E2 -13288.409} C_VEL
LIN {X 0,Y 354.789,Z 276.103,A -85,B 0,C 180,E1 -13291.619,E2 -13291.619} C_VEL
LIN {X 0,Y 354.825,Z 276.098,A -85,B 0,C 180,E1 -13295.661,E2 -13295.661} C_VEL
LIN {X 0,Y 354.819,Z 276.096,A -85,B 0,C 180,E1 -13299.117,E2 -13299.117} C_VEL
LIN {X 0,Y 354.998,Z 276.083,A -85,B 0,C 180,E1 -13302.564,E2 -13302.564} C_VEL
LIN {X 0,Y 354.949,Z 281.352,A -85,B 0,C 180,E1 -13303.954,E2 -13303.954} C_VEL
LIN {X 0,Y 357.594,Z 301.227,A -85,B 0,C 180,E1 -13304.575,E2 -13304.575} C_VEL
LIN {X 0,Y 356.396,Z 360.465,A -85,B 0,C 180,E1 -13306.207,E2 -13306.207} C_VEL
LIN {X 0,Y 356.159,Z 370.859,A -85,B 0,C 180,E1 -13306.67,E2 -13306.67} C_VEL
LIN {X 0,Y 355.816,Z 381.244,A -85,B 0,C 180,E1 -13307.311,E2 -13307.311} C_VEL
LIN {X 0,Y 355.476,Z 391.619,A -85,B 0,C 180,E1 -13308.168,E2 -13308.168} C_VEL
LIN {X 0,Y 355.034,Z 400.981,A -85,B 0,C 180,E1 -13309.165,E2 -13309.165} C_VEL
LIN {X 0,Y 354.645,Z 408.639,A -85,B 0,C 180,E1 -13310.163,E2 -13310.163} C_VEL
LIN {X 0,Y 354.208,Z 416.742,A -85,B 0,C 180,E1 -13311.446,E2 -13311.446} C_VEL
LIN {X 0,Y 353.947,Z 423.816,A -85,B 0,C 180,E1 -13312.875,E2 -13312.875} C_VEL
LIN {X 0,Y 353.667,Z 429.439,A -85,B 0,C 180,E1 -13314.302,E2 -13314.302} C_VEL
LIN {X 0,Y 353.603,Z 433.085,A -85,B 0,C 180,E1 -13315.444,E2 -13315.444} C_VEL
LIN {X 0,Y 353.387,Z 437.279,A -85,B 0,C 180,E1 -13317.154,E2 -13317.154} C_VEL
LIN {X 0,Y 353.339,Z 440.124,A -85,B 0,C 180,E1 -13318.864,E2 -13318.864} C_VEL
LIN {X 0,Y 353.368,Z 441.241,A -85,B 0,C 180,E1 -13320.004,E2 -13320.004} C_VEL
LIN {X 0,Y 353.433,Z 441.801,A -85,B 0,C 180,E1 -13321.143,E2 -13321.143} C_VEL
LIN {X 0,Y 353.569,Z 441.84,A -85,B 0,C 180,E1 -13322.282,E2 -13322.282} C_VEL
LIN {X 0,Y 353.835,Z 441.356,A -85,B 0,C 180,E1 -13323.42,E2 -13323.42} C_VEL
LIN {X 0,Y 354.126,Z 440.347,A -85,B 0,C 180,E1 -13324.557,E2 -13324.557} C_VEL
LIN {X 0,Y 354.356,Z 438.769,A -85,B 0,C 180,E1 -13325.695,E2 -13325.695} C_VEL
LIN {X 0,Y 354.411,Z 436.585,A -85,B 0,C 180,E1 -13326.837,E2 -13326.837} C_VEL
LIN {X 0,Y 355.284,Z 432.283,A -85,B 0,C 180,E1 -13328.478,E2 -13328.478} C_VEL
LIN {X 0,Y 355.939,Z 427.137,A -85,B 0,C 180,E1 -13329.952,E2 -13329.952} C_VEL
LIN {X 0,Y 356.823,Z 420.927,A -85,B 0,C 180,E1 -13331.363,E2 -13331.363} C_VEL
LIN {X 0,Y 357.919,Z 413.179,A -85,B 0,C 180,E1 -13332.765,E2 -13332.765} C_VEL
LIN {X 0,Y 358.975,Z 404.218,A -85,B 0,C 180,E1 -13334.024,E2 -13334.024} C_VEL
LIN {X 0,Y 359.869,Z 395.574,A -85,B 0,C 180,E1 -13335,E2 -13335} C_VEL
LIN {X 0,Y 360.878,Z 384.68,A -85,B 0,C 180,E1 -13335.97,E2 -13335.97} C_VEL
LIN {X 0,Y 361.686,Z 372.918,A -85,B 0,C 180,E1 -13336.731,E2 -13336.731} C_VEL
LIN {X 0,Y 362.327,Z 361.79,A -85,B 0,C 180,E1 -13337.245,E2 -13337.245} C_VEL
LIN {X 0,Y 364.828,Z 306.045,A -85,B 0,C 180,E1 -13338.961,E2 -13338.961} C_VEL
LIN {X 0,Y 362.139,Z 295.639,A -85,B 0,C 180,E1 -13339.616,E2 -13339.616} C_VEL
LIN {X 0,Y 358.065,Z 286.912,A -85,B 0,C 180,E1 -13340.395,E2 -13340.395} C_VEL
LIN {X 0,Y 357.145,Z 284.8,A -85,B 0,C 180,E1 -13340.583,E2 -13340.583} C_VEL
LIN {X 0,Y 354.83,Z 276.1,A -85,B 0,C 180,E1 -13343.464,E2 -13343.464} C_VEL
LIN {X 0,Y 354.816,Z 276.103,A -85,B 0,C 180,E1 -13347.105,E2 -13347.105} C_VEL
LIN {X 0,Y 354.806,Z 276.102,A -85,B 0,C 180,E1 -13349.686,E2 -13349.686} C_VEL
LIN {X 0,Y 354.796,Z 276.105,A -85,B 0,C 180,E1 -13352.335,E2 -13352.335} C_VEL
LIN {X 0,Y 354.828,Z 276.098,A -85,B 0,C 180,E1 -13355.7,E2 -13355.7} C_VEL
LIN {X 0,Y 354.778,Z 276.104,A -85,B 0,C 180,E1 -13359.414,E2 -13359.414} C_VEL
LIN {X 0,Y 354.795,Z 276.102,A -85,B 0,C 180,E1 -13362.868,E2 -13362.868} C_VEL
LIN {X 0,Y 354.777,Z 276.103,A -85,B 0,C 180,E1 -13366.105,E2 -13366.105} C_VEL
LIN {X 0,Y 354.794,Z 276.103,A -85,B 0,C 180,E1 -13369.18,E2 -13369.18} C_VEL
LIN {X 0,Y 354.811,Z 276.103,A -85,B 0,C 180,E1 -13372.405,E2 -13372.405} C_VEL
LIN {X 0,Y 354.821,Z 276.1,A -85,B 0,C 180,E1 -13374.941,E2 -13374.941} C_VEL
LIN {X 0,Y 354.803,Z 276.098,A -85,B 0,C 180,E1 -13378.406,E2 -13378.406} C_VEL
LIN {X 0,Y 354.858,Z 276.096,A -85,B 0,C 180,E1 -13381.619,E2 -13381.619} C_VEL
